Yaskawa INFORM job: KRIS7-TEST.JBI

/JOB
//NAME KRIS7-TEST
//POS
///NPOS 468,468,468,16,0,0
///TOOL 0
///POSTYPE PULSE
///PULSE
C00000=-36471,-76527,-106813,19264,71481,77238
C00001=-36471,-76527,-106813,19264,71481,77238
C00002=-63812,-119516,-80644,-27282,71106,59809
C00003=-86670,-29465,-24103,-33182,93398,46515
C00004=-88663,-31189,-25266,-33292,92471,45985
C00005=-89600,-31952,-25776,-33339,92036,45737
C00006=-88663,-31189,-25266,-33292,92471,45985
C00007=-88663,-31929,-28188,-33361,93666,45629
C00008=-101397,-33118,-34088,-22474,91022,41668
C00009=-101397,-32934,-33069,-22469,90527,41762
C00010=-101397,-33275,-35023,-22483,91481,41581
C00011=-104499,20623,14787,-23283,115207,62973
C00012=-104352,17765,12486,-23220,115200,63034
C00013=-104529,15851,10717,-23303,115245,62949
C00014=-104352,17765,12486,-23220,115200,63034
C00015=-100086,19810,13187,-22516,115799,63398
C00016=-93288,781,-1160,-33549,91987,44264
C00017=-95103,1586,-482,-33591,91265,43744
C00018=-95638,1156,-842,-33600,91054,43591
C00019=-95103,1586,-482,-33591,91265,43744
C00020=-100253,-3614,-11898,-25466,91372,41970
C00021=-107199,-8537,-17665,-19004,89460,40114
C00022=-108350,-8919,-17473,-17740,88760,39873
C00023=-102096,-5783,-13006,-25389,90415,41488
C00024=-93175,-13453,-24658,-25770,96080,43586
C00025=-29596,-126908,-80456,-16683,91164,67663
C00026=-130966,-130992,-81417,14801,93022,-34731
C00027=-139735,-123676,-71676,23223,79574,-40827
C00028=-136755,-124231,-71804,23689,78586,-39979
C00029=-134984,-124514,-71869,23951,78010,-39473
C00030=-136755,-124231,-71804,23689,78586,-39979
C00031=-136306,-124758,-74432,23664,79703,-39597
C00032=-105195,-127447,-79852,15126,73259,-28242
C00033=-104798,-126140,-77647,15190,72530,-28198
C00034=-108375,-128078,-79564,15067,73342,-29336
C00035=-112121,-93277,-65445,16297,96104,-47809
C00036=-116095,-84503,-58814,18813,102506,-48434
C00037=-114391,-86924,-59797,19239,101506,-47972
C00038=-116095,-84503,-58814,18813,102506,-48434
C00039=-117812,-129995,-81150,14641,74986,-32390
C00040=-118791,-92886,-67151,14205,85296,-31516
C00041=-116748,-92781,-67110,14299,84968,-30842
C00042=-115499,-92681,-67072,14351,84774,-30431
C00043=-116748,-92781,-67110,14299,84968,-30842
C00044=-116748,-94243,-70296,14285,86141,-30707
C00045=-102870,-92009,-70676,9222,86435,-25689
C00046=-102870,-90997,-68303,9229,85506,-25758
C00047=-102870,-92009,-70676,9222,86435,-25689
C00048=-124106,-98193,-79828,8318,91183,-32632
C00049=-120990,-117719,-86799,1028,78019,83969
C00050=-103618,-122878,-84450,6731,45671,69045
C00051=-107839,-39273,-43881,11021,86771,60654
C00052=-102663,-26959,-34255,5037,90909,61236
C00053=-106417,-22492,-30421,10624,98396,60708
C00054=-103076,-37240,-40581,8849,97261,61678
C00055=-110992,-39766,-43585,17340,97602,59383
C00056=-111851,-103912,-94699,10334,87868,68255
C00057=-100525,-93554,-87313,9422,87254,72087
C00058=-95765,-72558,-76889,7644,100510,59309
C00059=-95463,-76426,-71939,16938,115118,61391
C00060=-102124,-64154,-61473,23072,122501,60539
C00061=-108072,-63754,-61449,27079,123073,58329
C00062=-126453,-110744,-88068,25157,96958,85114
C00063=-124535,-114305,-86499,25277,93833,85163
C00064=-121951,-112497,-85625,25654,93398,86032
C00065=-116232,-108405,-84002,26384,92604,88006
C00066=-122754,-106725,-87203,25770,97209,86568
C00067=-142865,-91008,-85242,17891,113758,73123
C00068=-142005,-90205,-84914,18160,113770,73464
C00069=-93871,-48257,-54590,-14207,101968,-48555
C00070=-106716,17042,-5346,-15024,102835,-53222
C00071=-114740,-14345,-34597,-13608,101053,-59815
C00072=-127078,-3386,-21930,-8482,103399,-53955
C00073=-129021,-1243,-17298,-7607,102543,-53064
C00074=-129893,-13096,-22178,-14005,113849,-54571
C00075=-129597,-5294,-13720,-15224,118044,-55057
C00076=-122058,-3228,-13278,-23261,119236,-52777
C00077=-102997,28917,14853,-20600,116287,-84527
C00078=-102792,-6395,-13177,-23260,105514,-87254
C00079=-105472,-3384,-9862,-23514,105257,-88219
C00080=-107060,-2107,-8876,-23770,104848,-88744
C00081=-104416,1445,-8009,-23523,106791,-88129
C00082=-100743,5943,-9423,-11985,113108,-51981
C00083=-104100,-22795,-28366,-25068,61310,-50210
C00084=-122112,-33809,-21710,-17217,45375,-58941
C00085=-130767,-31374,-20493,-827,48037,-55558
C00086=-127443,-25046,-15801,-6227,47707,-53970
C00087=-124818,-6385,-1356,-9028,48013,-52772
C00088=-117469,-7945,-6130,-22808,51414,-49873
C00089=-27812,-119319,-87277,-42007,83182,-24370
C00090=-5621,-139291,-109992,-39952,96377,80222
C00091=-5621,-139291,-109992,-39952,96377,80222
C00092=87039,-115654,-82424,8022,52039,63522
C00093=129513,-144814,-136934,9080,53426,64546
C00094=125697,-42562,-22948,15669,36761,60413
C00095=126411,-45246,-5808,21270,25248,57573
C00096=137384,-94042,-14593,40484,4605,50802
C00097=156551,-106329,-15137,73999,-7456,40548
C00098=21972,-55240,6153,47914,22932,-29567
C00099=21236,-16271,22987,30471,58724,-17539
C00100=25572,-13994,24670,30139,57395,-16133
C00101=25572,-13994,24670,30139,57395,-16133
C00102=25572,-11360,29564,30679,55956,-16584
C00103=25572,-11642,29045,30620,56106,-16536
C00104=27131,-10690,29771,30483,55623,-16029
C00105=26687,-10968,29556,30524,55761,-16173
C00106=26687,-11435,28694,30427,56011,-16093
C00107=27498,-10924,29084,30350,55760,-15829
C00108=25574,-12112,28179,30521,56353,-16458
C00109=45065,-62251,-3802,30710,44756,-11744
C00110=45065,-62251,-3802,30710,44756,-11744
C00111=45062,-59455,603,31381,43658,-12167
C00112=45063,-59751,140,31308,43771,-12121
C00113=47363,-58455,705,30723,43318,-11195
C00114=46715,-58835,536,30894,43443,-11458
C00115=46717,-59324,-234,30775,43632,-11382
C00116=47899,-58629,71,30459,43407,-10903
C00117=45070,-60247,-636,31184,43956,-12046
C00118=91239,-86156,-11635,17290,26072,6257
C00119=91239,-86156,-11635,17290,26072,6257
C00120=91235,-83004,-7277,17966,25059,5922
C00121=91238,-83335,-7734,17887,25164,5961
C00122=92915,-81478,-7301,16273,25546,7147
C00123=92456,-82017,-7434,16717,25431,6822
C00124=92461,-82561,-8193,16597,25608,6883
C00125=93295,-81576,-7954,15794,25823,7471
C00126=91253,-83887,-8499,17745,25338,6030
C00127=158815,-84367,-11225,-29167,32105,45030
C00128=158815,-84367,-11225,-29167,32105,45030
C00129=158813,-81248,-6866,-30028,31158,45482
C00130=158816,-81574,-7323,-29937,31259,45435
C00131=156798,-79782,-6873,-28651,31269,44264
C00132=157356,-80302,-7010,-29015,31259,44592
C00133=157361,-80840,-7770,-28870,31430,44517
C00134=156355,-79886,-7523,-28212,31458,43925
C00135=158825,-82117,-8087,-29789,31433,45356
C00136=202470,-53277,302,-32057,53464,57737
C00137=202470,-53277,302,-32057,53464,57737
C00138=202470,-50579,4744,-32592,52316,58142
C00139=202471,-50863,4277,-32535,52437,58099
C00140=200347,-49670,4876,-32326,51937,57354
C00141=200948,-50019,4697,-32389,52078,57566
C00142=200949,-50488,3922,-32295,52282,57496
C00143=199855,-49845,4246,-32177,52030,57107
C00144=202472,-51331,3500,-32439,52645,58024
C00145=129513,-144814,-136934,9080,53426,64546
C00146=129513,-144814,-136934,9080,53426,64546
C00147=129513,-109632,-69732,14359,30578,61412
C00148=129513,-83278,-28536,22379,19314,57484
C00149=122399,-55102,-4999,-8402,35911,61097
C00150=119920,-45288,5620,-7331,30390,60229
C00151=119750,-46058,4611,-7150,30605,60108
C00152=119750,-45110,6218,-7257,30106,60163
C00153=119736,-46268,4531,-7151,30546,60106
C00154=119736,-47979,3777,-7238,30135,60151
C00155=119727,-46869,5444,-7329,29678,60198
C00156=119739,-46062,5830,-7299,29854,60181
C00157=119715,-47768,4014,-7231,30094,60141
C00158=122330,-55612,-6297,-8657,32618,61353
C00159=121709,-73745,-24049,9098,30676,53116
C00160=129398,-114812,-46545,3278,22913,57364
C00161=129398,-114812,-46545,3278,22913,57364
C00162=147189,-126166,-80752,5474,34460,60082
C00163=165214,-137669,-115409,7698,46160,62836
C00164=176409,-144814,-136934,9080,53426,64546
C00165=176409,-109327,-69248,14418,30440,61382
C00166=137996,-109327,-69248,14418,30440,61382
C00167=136854,5077,41656,21727,21645,57624
C00168=123203,14789,51546,53172,38991,40073
C00169=123077,34948,78392,59944,35543,36223
C00170=123077,37993,83408,61838,34770,35183
C00171=123098,35348,79007,60153,35442,36112
C00172=123139,31348,74887,59568,35673,36443
C00173=123149,34907,80133,61289,34946,35499
C00174=123130,37074,82445,61677,34805,35280
C00175=123183,30422,73312,58971,35912,36781
C00176=123599,57381,99984,51632,43856,40437
C00177=128629,59731,102899,52063,41097,41453
C00178=130023,30320,69348,52154,35987,38987
C00179=132104,19481,50493,23737,37003,47692
C00180=136200,48792,78585,9333,46433,53780
C00181=127667,43842,73216,11867,48213,50363
C00182=127110,36942,61073,12684,52130,50324
C00183=125174,17943,48073,21449,38985,45601
C00184=109988,7135,45797,56276,48109,34557
C00185=110783,-2370,26113,10588,43916,42309
C00186=96618,15106,36280,16308,48845,36588
C00187=99195,57631,83562,8929,54990,39222
C00188=83229,75338,108095,18392,45531,30732
C00189=82057,52050,70954,17595,54461,31693
C00190=99279,-29834,2408,12633,51480,38376
C00191=124602,-34297,-476,3581,48489,48797
C00192=129000,-155474,-110821,1722,53982,50766
C00193=129000,-186332,-136923,1718,54189,50769
C00194=129000,-186332,-136923,1718,54189,50769
C00195=124634,-42983,-17396,3288,54424,49011
C00196=119975,43106,65207,5416,48088,46799
C00197=124227,21838,45287,-4126,60993,49348
C00198=115102,22260,45694,-2630,60591,46004
C00199=111900,23179,46586,-2094,60423,44829
C00200=106599,25422,48781,-1196,60121,42879
C00201=109500,51617,73450,-2873,46958,44240
C00202=119708,-19564,1692,5024,54962,47046
C00203=124398,4257,31803,38326,49723,41965
C00204=124500,-5455,16693,36249,53145,43496
C00205=123978,22175,41893,32824,63757,46964
C00206=136633,26599,46213,31259,58773,50852
C00207=137127,47274,64261,33367,46328,47205
C00208=127043,-60461,-47717,31537,61680,47716
C00209=130427,-104246,-66216,34447,50964,45598
C00210=130427,-131180,-133049,27346,74705,52630
C00211=129293,-131648,-133187,27764,74930,52255
C00212=129293,-112975,-80869,32941,55210,46617
C00213=125224,-26758,-13299,33226,59088,46051
C00214=97492,-17863,6740,47317,62068,35221
C00215=76763,21057,43225,48272,71101,29312
C00216=80709,51150,75439,39481,73131,33496
C00217=101893,22474,45257,39781,66883,40263
C00218=98002,-1326,18556,46821,62661,35806
C00219=97492,-17863,6740,47317,62068,35221
C00220=125224,-26758,-13299,33226,59088,46051
C00221=129293,-131648,-133187,27764,74930,52255
C00222=129293,-130373,-135142,27565,76585,52657
C00223=129293,-130373,-135142,27565,76585,52657
C00224=129293,-130373,-135142,27565,76585,52657
C00225=126775,-65943,-41926,33631,56357,45828
C00226=146499,-5820,8509,-12483,47348,74367
C00227=133227,18598,33392,-5127,43166,68552
C00228=134087,40556,59352,-4333,44134,68757
C00229=109518,39473,58200,8432,44907,57480
C00230=110804,22133,33080,8574,45677,58038
C00231=95832,-100308,-60228,18401,42759,50383
C00232=85717,-180836,-128237,23276,45701,46095
C00233=134324,-194207,-130804,-6935,34984,69726
C00234=134324,-194207,-130804,-6935,34984,69726
C00235=134324,-194207,-130804,-6935,34984,69726
C00236=126554,-62104,-55568,-768,56192,65237
C00237=102691,-29899,-32559,11070,60126,55987
C00238=93699,-1684,15739,18283,46963,50224
C00239=95177,34388,59282,20423,38809,49091
C00240=95427,37375,44105,11480,58003,52927
C00241=82804,57701,66332,15963,56969,47713
C00242=80078,42075,52490,24500,50349,44630
C00243=92595,-4722,8571,18053,49920,50291
C00244=90890,13188,28851,45241,66990,53478
C00245=96516,51970,78121,48970,56932,51018
C00246=108766,35550,55769,36284,51974,56943
C00247=109501,48300,76470,39344,46724,54946
C00248=112089,47430,75488,38680,45769,55875
C00249=109461,35195,57508,36711,50675,56747
C00250=102961,43860,64049,37370,53600,54832
C00251=117347,37004,56694,33344,48695,60037
C00252=107165,27849,47408,45061,56134,56400
C00253=93699,-1684,15739,18283,46963,50224
C00254=126554,-62104,-55568,-768,56192,65237
C00255=132741,-190295,-136907,-5065,40605,68463
C00256=132741,-190295,-136907,-5065,40605,68463
C00257=132741,-190295,-136907,-5065,40605,68463
C00258=132741,-190295,-136907,-5065,40605,68463
C00259=126216,-48827,-32555,-652,48851,65144
C00260=116157,12397,26645,-836,43828,61032
C00261=107201,15073,29086,4732,43915,56787
C00262=108708,45240,59560,984,53519,57995
C00263=105889,47117,61614,1966,53270,56850
C00264=104117,15965,27840,6481,45345,55424
C00265=116157,12397,26645,-836,43828,61032
C00266=115184,32776,48658,-853,48273,60616
C00267=102009,39914,56094,5283,47719,54846
C00268=104295,38849,56164,-3583,45498,56420
C00269=106773,10666,21679,-1556,45201,57174
C00270=121513,8451,23347,32656,44981,60126
C00271=121479,33249,54130,32703,45073,60132
C00272=136244,38436,59676,26271,39414,66032
C00273=133358,13884,30500,26959,39421,64637
C00274=126216,-48827,-32555,-652,48851,65144
C00275=132741,-190295,-136907,-5065,40605,68463
C00276=132741,-190295,-136907,-5065,40605,68463
C00277=132741,-190295,-136907,-5065,40605,68463
C00278=132741,-190295,-136907,-5065,40605,68463
C00279=126554,-62104,-55568,-768,56192,65237
C00280=93699,-1684,15739,18283,46963,50224
C00281=109219,22842,33799,17593,55341,60017
C00282=114933,32716,55729,7970,41115,61622
C00283=98115,43367,67193,11592,40390,54327
C00284=92675,33947,50979,20393,49569,52577
C00285=113935,26100,44118,24451,47496,60162
C00286=114558,35388,59860,26260,42851,59091
C00287=117732,34768,59212,24806,41998,60459
C00288=114305,24559,43264,24398,47147,60243
C00289=99844,11402,27037,25299,53213,55440
C00290=126554,-62104,-55568,-768,56192,65237
C00291=132741,-190295,-136907,-5065,40605,68463
C00292=132741,-190295,-136907,-5065,40605,68463
C00293=132741,-190295,-136907,-5065,40605,68463
C00294=132741,-190295,-136907,-5065,40605,68463
C00295=126216,-48827,-32555,-652,48851,65144
C00296=134748,7082,18366,-200,46227,68791
C00297=132038,36511,51354,2924,49864,67481
C00298=110399,36003,50767,11764,51912,58463
C00299=101806,27679,40045,16592,51225,54569
C00300=102258,33237,49963,17192,48019,54198
C00301=104874,31614,48575,4374,45128,56525
C00302=106858,16986,29459,6761,48587,57166
C00303=113156,-2573,6178,11839,50347,59373
C00304=100847,-116604,-69788,21646,41420,51852
C00305=93537,-194381,-130385,26473,40988,47897
C00306=104459,-185785,-128899,13362,14722,54877
C00307=137185,-168918,-120422,-22616,31853,56508
C00308=103466,-143035,-89833,18127,44217,-664
C00309=153034,-42791,-3789,-574,51224,21077
C00310=154411,-23786,22188,6392,45845,11810
C00311=163692,-14831,30793,3045,43978,15753
C00312=162658,-12144,32796,3380,44162,15317
C00313=162658,-10372,35929,3443,43146,15280
C00314=162658,-10822,35136,3427,43403,15291
C00315=163644,-13399,33193,3102,43239,15709
C00316=163644,-12612,34572,3127,42795,15690
C00317=163043,-11060,35746,3327,42891,15434
C00318=163515,-12286,34819,3170,42815,15635
C00319=166152,-32133,5550,1997,50546,16952
C00320=100006,-46830,-3879,17345,57754,-8477
C00321=55652,-4276,24712,7053,56203,-22524
C00322=50070,19037,58848,16400,45172,-27179
C00323=51341,29328,71603,16783,42484,-27133
C00324=51341,32600,77102,17341,40853,-27469
C00325=51341,31422,75137,17137,41430,-27347
C00326=50264,28853,72458,17349,41942,-27728
C00327=50264,30492,75208,17635,41129,-27900
C00328=50738,31631,76404,17545,40896,-27733
C00329=50419,30858,75590,17605,41054,-27844
C00330=50419,14018,45638,14959,50461,-26136
C00331=53903,-12653,21571,13778,50962,-24612
C00332=66094,-67687,-18476,10677,45688,-20127
C00333=87454,-109874,-47340,-27972,40441,7116
C00334=78946,-55292,-6224,-23492,40558,2756
C00335=70027,-40972,10385,-20890,35738,-464
C00336=63439,-31094,22495,-18522,32104,-3061
C00337=63439,-29243,25592,-19018,31198,-2801
C00338=75556,-28394,37292,-62320,27769,16956
C00339=74155,-27422,37887,-61985,27131,16453
C00340=64318,-30449,24372,-21159,31089,-1672
C00341=67917,-25293,27676,-22824,32488,-51
C00342=67917,-25293,27676,-22824,32488,-51
C00343=68696,-24050,28500,-23162,32795,289
C00344=67917,-25293,27676,-22824,32488,-51
C00345=75368,-51805,-10970,-21451,43738,562
C00346=86139,-25078,5298,-24076,50017,4008
C00347=83917,-18337,16451,-24570,46284,3982
C00348=79836,-11066,25880,-23931,43276,2865
C00349=79836,-9413,28995,-24399,42297,3151
C00350=86314,-11086,32289,-42271,40319,10375
C00351=84998,-9998,33124,-41890,39785,9892
C00352=80963,-11349,26642,-26884,42529,4054
C00353=82363,-6834,30155,-27320,43093,4575
C00354=82761,-5465,31244,-27447,43243,4725
C00355=83186,-3958,32457,-27584,43396,4888
C00356=82761,-5465,31244,-27447,43243,4725
C00357=87385,-23200,183,-25112,53654,3858
C00358=88611,-6659,17671,-26227,51974,4862
C00359=85936,239,26154,-25964,49655,4281
C00360=85936,1480,28752,-26325,48787,4530
C00361=91127,630,32748,-40408,46738,9768
C00362=90313,1326,33333,-40211,46382,9497
C00363=86792,7,26768,-28149,49107,5083
C00364=90602,-33059,-4237,-28517,52203,5912
C00365=94576,-67258,-23025,57506,77870,-531
C00366=122383,-58832,-3556,65417,58097,774
C00367=127343,-13643,25366,63114,57669,4189
C00368=131296,13324,53885,65824,53660,3026
C00369=131296,14618,56173,66322,53341,2642
C00370=130824,14275,55697,67245,54004,2465
C00371=131723,14569,55971,67399,53464,2593
C00372=130860,14268,55674,67244,53987,2476
C00373=127124,-5804,29633,63377,58737,4694
C00374=126701,-15037,22522,63119,61223,3769
C00375=126701,1136,51385,68187,57095,-774
C00376=131284,6353,59362,70779,53649,-1335
C00377=131284,8754,63319,71617,53230,-1977
C00378=131284,6353,59362,70779,53649,-1335
C00379=132452,6685,59657,71098,52984,-1198
C00380=131284,6353,59362,70779,53649,-1335
C00381=131052,11501,64001,70861,53706,-1474
C00382=130893,14100,66417,70922,53742,-1574
C00383=130719,17099,69269,71021,53763,-1708
C00384=130893,14100,66417,70922,53742,-1574
C00385=128315,-22064,27147,66784,57381,941
C00386=129627,-37207,17556,68184,55855,186
C00387=130148,-23471,44300,74760,52317,-4741
C00388=135320,-14449,56479,79067,48853,-5949
C00389=135320,-12066,60154,79963,48630,-6563
C00390=135320,-14449,56479,79067,48853,-5949
C00391=137070,-14043,56767,79770,47945,-5809
C00392=135320,-14449,56479,79067,48853,-5949
C00393=134716,-10676,59212,78597,49226,-5841
C00394=134466,-8976,60486,78417,49378,-5807
C00395=134182,-6930,62050,78227,49545,-5776
C00396=134466,-8976,60486,78417,49378,-5807
C00397=106496,-51026,-9475,59829,73743,881
C00398=106496,-62277,-31108,58328,77765,3910
C00399=137468,-45448,-13164,23993,62707,9546
C00400=142031,-34381,-3630,18745,59946,9254
C00401=153480,-23481,18954,7895,48240,10284
C00402=154576,-15419,32985,7624,43640,10304
C00403=154522,-15140,33190,7639,43662,10282
C00404=163868,-10589,37972,6252,39486,12143
C00405=163705,-4288,45034,21073,38117,2051
C00406=163923,-2936,48273,26703,35302,170
C00407=146970,-27557,19782,29282,44621,-5055
C00408=77984,-28544,12598,9594,52255,-4511
C00409=87028,-14899,33509,-8097,43242,2023
C00410=86974,-14913,33498,-8080,43236,2001
C00411=77485,-7266,39372,-4959,42873,-2067
C00412=74579,-2521,47308,-17915,35684,548
C00413=75615,102,52227,-26296,32839,3633
C00414=84696,-19604,28451,-27180,39406,6073
C00415=87454,-109874,-47340,-27972,40441,7116
C00416=87454,-109874,-47340,-27972,40441,7116
C00417=73980,-36973,3355,-18473,60366,27525
C00418=58877,-27993,19766,-16405,50257,19650
C00419=71120,-6285,35203,-17245,53240,22132
C00420=69479,-8808,33067,-14788,50723,16894
C00421=73605,-31096,1389,-14177,59206,17320
C00422=72431,-18207,17991,-16956,51529,14828
C00423=73562,-15726,19761,-17396,52120,15565
C00424=83313,14185,44247,-21039,56473,22237
C00425=84211,-11070,13701,-18734,53182,26231
C00426=82998,-523,24465,-18637,51768,25979
C00427=82448,-570,28041,-15362,40529,26924
C00428=77134,-2165,39833,11119,14146,19838
C00429=76844,-12553,31864,7458,12108,20601
C00430=84341,-54767,463,-16268,10060,32559
C00431=79893,-46463,9240,-49361,8484,37720
C00432=71243,-22477,30789,30336,5200,-490
C00433=70979,-19028,33557,31433,5346,-1026
C00434=68683,-10375,50772,112552,4351,-37626
C00435=72976,-34040,25530,30096,2440,-170
C00436=51638,-47354,18402,88201,13764,-30312
C00437=50365,-30767,37744,101133,14655,-36527
C00438=46532,-17600,60099,119714,18815,-46088
C00439=50533,-52861,21550,106572,14840,-38992
C00440=66288,-93178,-46103,5866,60369,16168
C00441=112510,-98188,-44790,18471,62864,-44268
C00442=149625,-37879,6780,17046,57011,-35751
C00443=155605,-32525,16928,15112,50177,-29308
C00444=149418,-7594,34122,13784,51545,-27133
C00445=143716,-10385,36525,25765,46016,-27057
C00446=147766,-22217,9496,11268,57983,-23560
C00447=146875,-12758,20894,15319,55227,-24771
C00448=146053,-8471,24161,15451,55560,-25047
C00449=142035,19351,48051,16301,55907,-26583
C00450=141803,14161,44980,18392,51510,-21349
C00451=142040,5818,24378,13474,61789,-22474
C00452=138840,15265,37176,20739,58625,-24937
C00453=138706,17261,38894,20771,58629,-24991
C00454=139526,10572,40705,23596,37058,-29346
C00455=140566,11430,47120,26457,25355,-31911
C00456=140419,-8993,28489,25719,26277,-31573
C00457=142059,-17553,21658,25375,25949,-31323
C00458=143624,-11159,28730,24740,24544,-30775
C00459=144392,-5853,43056,31020,18891,-33660
C00460=150093,-42733,14524,24992,16002,-29807
C00461=146967,-32270,24662,40502,20136,-34953
C00462=144755,-20255,35089,33636,31779,-30408
C00463=144236,-61611,5153,41773,14596,-38681
C00464=136995,-150356,-85047,33892,64386,-36535
C00465=136995,-178339,-110283,33604,8697,-36217
C00466=130728,-161100,-136081,16173,33339,-28558
C00467=1271,-161100,-136081,16173,33339,-28558
BC00000=295325,674563,1075170
BC00001=295325,674563,1075170
BC00002=396971,731967,797664
BC00003=396971,731967,797664
BC00004=396971,731967,797664
BC00005=396971,731967,797664
BC00006=396971,731967,797664
BC00007=396971,731967,797664
BC00008=396971,731967,797664
BC00009=396971,731967,797664
BC00010=396971,731967,797664
BC00011=396971,731967,797664
BC00012=396971,731967,797664
BC00013=396971,731967,797664
BC00014=396971,731967,797664
BC00015=396971,731967,797664
BC00016=396971,731967,797664
BC00017=396971,731967,797664
BC00018=396971,731967,797664
BC00019=396971,731967,797664
BC00020=396971,731967,797664
BC00021=396971,731967,797664
BC00022=396971,731967,797664
BC00023=396971,731967,797664
BC00024=396971,731967,797664
BC00025=396971,731967,797664
BC00026=1331,731967,797664
BC00027=1331,834817,797664
BC00028=1331,834817,797664
BC00029=1331,834817,797664
BC00030=1331,834817,797664
BC00031=1331,834817,797664
BC00032=1331,834817,797664
BC00033=1331,834817,797664
BC00034=1331,834817,797664
BC00035=1331,834817,797664
BC00036=1331,834817,797664
BC00037=1331,834817,797664
BC00038=1331,834817,797664
BC00039=1331,834817,797664
BC00040=1331,834817,797664
BC00041=1331,834817,797664
BC00042=1331,834817,797664
BC00043=1331,834817,797664
BC00044=1331,834817,797664
BC00045=1331,834817,797664
BC00046=1331,834817,797664
BC00047=1331,834817,797664
BC00048=1331,834817,797664
BC00049=1072,761065,516765
BC00050=1072,827865,516765
BC00051=1071,829671,517043
BC00052=1071,829895,517078
BC00053=1071,829895,517078
BC00054=1071,829895,517078
BC00055=1071,829895,517078
BC00056=768,829895,695080
BC00057=768,829895,695080
BC00058=768,829895,695080
BC00059=768,829895,695080
BC00060=768,829895,695080
BC00061=768,829895,695080
BC00062=768,829895,695080
BC00063=768,829895,695080
BC00064=768,829895,695080
BC00065=768,829895,695080
BC00066=768,829895,695080
BC00067=768,829895,695080
BC00068=768,686767,695080
BC00069=396971,681851,797664
BC00070=396971,731967,797664
BC00071=396971,731967,797664
BC00072=396971,731967,797664
BC00073=396971,731967,797664
BC00074=396971,731967,797664
BC00075=396971,731967,797664
BC00076=396971,731967,797664
BC00077=396971,731967,797664
BC00078=396971,731967,797664
BC00079=396971,731967,797664
BC00080=396971,731967,797664
BC00081=396971,731967,797664
BC00082=396971,731967,797664
BC00083=396971,731967,516765
BC00084=396971,731967,516765
BC00085=396971,731967,516765
BC00086=396972,731979,516765
BC00087=396971,731967,516765
BC00088=396971,731967,516765
BC00089=396971,731967,516765
BC00090=188286,731967,1013423
BC00091=188286,774486,1052805
BC00092=125948,1177450,1071719
BC00093=215453,1309115,984509
BC00094=215453,1309115,984509
BC00095=215453,1269749,984509
BC00096=215453,1189879,984509
BC00097=215453,1164125,984509
BC00098=215453,1164125,984509
BC00099=215453,1164125,984509
BC00100=215453,1164125,984509
BC00101=215453,1164125,984509
BC00102=215453,1164125,984509
BC00103=215453,1164125,984509
BC00104=215453,1164125,984509
BC00105=215453,1164125,984509
BC00106=215453,1164125,984509
BC00107=215453,1164125,984509
BC00108=215453,1164125,984509
BC00109=215453,1164125,984509
BC00110=215453,1164125,984509
BC00111=215453,1164125,984509
BC00112=215453,1164125,984509
BC00113=215453,1164125,984509
BC00114=215453,1164125,984509
BC00115=215453,1164125,984509
BC00116=215453,1164125,984509
BC00117=215453,1164125,984509
BC00118=215453,1164125,984509
BC00119=215453,1164125,984509
BC00120=215453,1164125,984509
BC00121=215453,1164125,984509
BC00122=215453,1164125,984509
BC00123=215453,1164125,984509
BC00124=215453,1164125,984509
BC00125=215453,1164125,984509
BC00126=215453,1164125,984509
BC00127=215453,1164125,984509
BC00128=215453,1164125,984509
BC00129=215453,1164125,984509
BC00130=215453,1164125,984509
BC00131=215453,1164125,984509
BC00132=215453,1164125,984509
BC00133=215453,1164125,984509
BC00134=215453,1164125,984509
BC00135=215453,1164125,984509
BC00136=215453,1164125,984509
BC00137=215453,1164125,984509
BC00138=215453,1164125,984509
BC00139=215453,1164125,984509
BC00140=215453,1164125,984509
BC00141=215453,1164125,984509
BC00142=215453,1164125,984509
BC00143=215453,1164125,984509
BC00144=215453,1164125,984509
BC00145=215453,1309115,984509
BC00146=345399,1357897,984509
BC00147=345399,1357897,984509
BC00148=345399,1230997,984509
BC00149=346767,1230997,984506
BC00150=346767,1230997,984506
BC00151=346767,1230997,984506
BC00152=346767,1230997,984506
BC00153=346767,1230997,984506
BC00154=346767,1230997,984506
BC00155=346767,1230997,984506
BC00156=346767,1230997,984506
BC00157=346767,1230997,984506
BC00158=346767,1230997,984506
BC00159=309515,1253158,984507
BC00160=309515,1253158,984507
BC00161=309515,1328360,1051553
BC00162=314470,1361455,1064018
BC00163=253389,1357693,1050986
BC00164=215453,1309115,984509
BC00165=215453,1309115,984509
BC00166=135997,1309115,984509
BC00167=135997,1309115,984509
BC00168=135997,1309115,984509
BC00169=135997,1309115,984505
BC00170=135997,1309115,984505
BC00171=135997,1309115,984505
BC00172=135997,1309115,984505
BC00173=135997,1309115,984505
BC00174=135997,1309115,984505
BC00175=135997,1309115,984505
BC00176=135997,1309115,984509
BC00177=135997,1309115,984509
BC00178=135997,1309115,984509
BC00179=135997,1309115,984509
BC00180=135997,1309115,984509
BC00181=135997,1309115,984509
BC00182=135997,1309115,984509
BC00183=135997,1309115,984509
BC00184=135997,1309115,984509
BC00185=135997,1309115,984509
BC00186=94463,1309115,955550
BC00187=94463,1309115,963176
BC00188=94463,1309115,963176
BC00189=94463,1309115,963176
BC00190=94463,1309115,963176
BC00191=141941,1309115,963176
BC00192=141941,1309115,963176
BC00193=223116,1330631,963176
BC00194=328548,1330631,963176
BC00195=328548,1330631,963176
BC00196=328548,1330631,963176
BC00197=328548,1285890,963176
BC00198=328548,1285890,963176
BC00199=328548,1285890,963176
BC00200=328548,1285890,963176
BC00201=328548,1330631,963176
BC00202=328548,1291307,959498
BC00203=328548,1293601,963176
BC00204=328548,1288886,905196
BC00205=328548,1288886,905196
BC00206=328548,1288886,905196
BC00207=328824,1330631,905196
BC00208=328824,1330631,905196
BC00209=328824,1330631,905196
BC00210=328824,1330631,905196
BC00211=151003,1330631,905196
BC00212=151003,1330631,905196
BC00213=151003,1330631,905196
BC00214=103648,1289163,905196
BC00215=103648,1289163,905196
BC00216=103648,1289163,905196
BC00217=103648,1289163,905196
BC00218=103648,1289163,905196
BC00219=103648,1289163,905196
BC00220=151003,1330631,905196
BC00221=151003,1330631,905196
BC00222=151003,1330631,905196
BC00223=303803,1330631,905196
BC00224=303803,1330631,763831
BC00225=303803,1330631,902112
BC00226=303803,1330631,902112
BC00227=303803,1330631,902112
BC00228=303803,1330631,902112
BC00229=303803,1330631,902112
BC00230=303803,1330631,902112
BC00231=303803,1330631,902112
BC00232=303803,1330631,1003127
BC00233=236612,1330631,1003127
BC00234=137483,1330631,1003127
BC00235=136337,1325904,719417
BC00236=136337,1325904,818715
BC00237=87820,1325904,842743
BC00238=87820,1325904,951848
BC00239=87820,1325904,951848
BC00240=87820,1320020,844218
BC00241=87820,1320020,844218
BC00242=87820,1325904,927335
BC00243=87820,1325904,927335
BC00244=87820,1325904,927335
BC00245=87820,1325904,927335
BC00246=87820,1325904,927335
BC00247=87820,1325904,927335
BC00248=87820,1325904,927335
BC00249=87820,1325904,927335
BC00250=87820,1325904,890762
BC00251=87820,1325904,890392
BC00252=87820,1325904,927335
BC00253=87820,1325904,951848
BC00254=136337,1325904,818715
BC00255=136337,1325904,818715
BC00256=136337,1325904,998300
BC00257=310720,1325904,998300
BC00258=310720,1325904,777065
BC00259=310720,1325904,891809
BC00260=310720,1325904,891809
BC00261=310720,1325904,891809
BC00262=310720,1325904,891809
BC00263=310720,1325904,891809
BC00264=310720,1325904,891809
BC00265=310720,1325904,891809
BC00266=310720,1325904,891809
BC00267=310720,1325904,891809
BC00268=310720,1325904,891809
BC00269=310720,1325904,891809
BC00270=310720,1325904,891809
BC00271=310720,1325904,891809
BC00272=310720,1325904,891809
BC00273=310720,1325904,891809
BC00274=310720,1325904,891809
BC00275=310720,1325904,777065
BC00276=310720,1325904,998300
BC00277=136337,1325904,998300
BC00278=136337,1325904,818715
BC00279=136337,1325904,818715
BC00280=87820,1325904,951848
BC00281=87820,1325904,927335
BC00282=87820,1325904,927335
BC00283=87820,1325904,927335
BC00284=87820,1325904,927335
BC00285=87820,1325904,927335
BC00286=87820,1325904,927335
BC00287=87820,1325904,927335
BC00288=87820,1325904,927335
BC00289=87820,1325904,927335
BC00290=136337,1325904,818715
BC00291=136337,1325904,818715
BC00292=136337,1325904,998300
BC00293=310720,1325904,998300
BC00294=310720,1325904,777065
BC00295=310720,1325904,891809
BC00296=310720,1325904,891809
BC00297=310720,1325904,891809
BC00298=310720,1325904,891809
BC00299=310720,1325904,891809
BC00300=310720,1325904,891809
BC00301=310720,1325904,891809
BC00302=310720,1325904,891809
BC00303=310720,1325904,891809
BC00304=310720,1325904,891809
BC00305=310720,1325904,1051225
BC00306=230237,1331507,1051225
BC00307=214487,1257960,1051225
BC00308=187930,1133951,1051225
BC00309=187930,1063861,1051225
BC00310=187930,1063861,1051225
BC00311=187931,1063862,1051199
BC00312=187931,1063862,1051199
BC00313=187931,1063862,1051199
BC00314=187931,1063862,1051199
BC00315=187931,1063862,1051199
BC00316=187931,1063862,1051199
BC00317=187931,1063862,1051199
BC00318=187931,1063862,1051199
BC00319=187931,1063862,1051199
BC00320=187930,1063861,1051225
BC00321=187930,1063861,1051225
BC00322=187930,1063861,1051225
BC00323=187930,1063861,1051225
BC00324=187930,1063861,1051225
BC00325=187930,1063861,1051225
BC00326=187930,1063861,1051225
BC00327=187930,1063861,1051225
BC00328=187930,1063861,1051225
BC00329=187930,1063861,1051225
BC00330=187930,1063861,1051225
BC00331=187930,1063861,1051225
BC00332=187930,1063861,1051225
BC00333=244084,1125149,1051225
BC00334=244084,1125149,1051225
BC00335=244084,1125149,1051225
BC00336=244084,1125149,1051225
BC00337=244084,1125149,1051225
BC00338=244084,1125149,1051225
BC00339=244084,1125149,1051225
BC00340=244084,1125149,1051225
BC00341=244084,1125149,1051225
BC00342=244084,1125149,1051225
BC00343=244084,1125149,1051225
BC00344=244084,1125149,1051225
BC00345=244084,1125149,1051225
BC00346=244084,1125149,1051225
BC00347=244084,1125149,1051225
BC00348=244084,1125149,1051225
BC00349=244084,1125149,1051225
BC00350=244084,1125149,1051225
BC00351=244084,1125149,1051225
BC00352=244084,1125149,1051225
BC00353=244084,1125149,1051225
BC00354=244084,1125149,1051225
BC00355=244084,1125149,1051225
BC00356=244084,1125149,1051225
BC00357=244084,1125149,1051225
BC00358=244084,1125149,1051225
BC00359=244083,1125149,1051222
BC00360=244083,1125149,1051222
BC00361=244083,1125149,1051222
BC00362=244083,1125149,1051222
BC00363=244083,1125149,1051222
BC00364=244083,1125149,1051222
BC00365=244083,1125148,1051219
BC00366=166173,1125148,1051219
BC00367=166173,1125148,1051219
BC00368=166173,1142192,1051219
BC00369=166173,1142192,1051219
BC00370=166173,1142192,1051219
BC00371=166173,1142192,1051219
BC00372=166173,1142192,1051219
BC00373=166173,1142192,1051219
BC00374=166173,1142192,1051219
BC00375=166173,1142192,1051219
BC00376=166173,1142192,1051219
BC00377=166173,1142192,1051219
BC00378=166173,1142192,1051219
BC00379=166173,1142192,1051219
BC00380=166173,1142192,1051219
BC00381=166173,1142192,1051219
BC00382=166173,1142192,1051219
BC00383=166173,1142192,1051219
BC00384=166173,1142192,1051219
BC00385=166173,1142192,1051219
BC00386=166173,1142192,1051219
BC00387=166173,1142192,1051219
BC00388=166173,1142192,1051219
BC00389=166173,1142192,1051219
BC00390=166173,1142192,1051219
BC00391=166173,1142192,1051219
BC00392=166173,1142192,1051219
BC00393=166173,1142192,1051219
BC00394=166173,1142192,1051219
BC00395=166173,1142192,1051219
BC00396=166173,1142192,1051219
BC00397=166173,1142192,1051219
BC00398=166173,1142192,1051219
BC00399=180177,1091773,1051223
BC00400=182943,1081815,1051224
BC00401=187709,1064658,1051225
BC00402=187930,1063861,1051225
BC00403=187930,1063861,1051225
BC00404=187930,1063861,1051225
BC00405=187930,1063861,1051225
BC00406=187930,1063861,1051225
BC00407=187930,1063861,1051225
BC00408=244084,1063861,1051225
BC00409=244084,1063861,1051225
BC00410=244084,1063861,1051225
BC00411=244084,1063861,1051225
BC00412=244084,1063861,1051225
BC00413=244084,1063861,1051225
BC00414=244084,1063861,1051225
BC00415=244084,1063861,1051225
BC00416=244084,1125149,1051225
BC00417=244084,1125149,1051225
BC00418=244084,1125149,1051225
BC00419=244084,1125149,1051225
BC00420=244084,1125149,1051225
BC00421=244084,1125149,1051225
BC00422=244084,1125149,1051225
BC00423=244084,1125149,1051225
BC00424=244084,1125149,1051225
BC00425=244084,1125149,1051225
BC00426=244084,1125149,1051225
BC00427=244084,1125149,1051225
BC00428=244084,1125149,1051225
BC00429=244084,1125149,1051225
BC00430=244084,1125149,1051225
BC00431=244084,1125149,1051225
BC00432=244084,1125149,1051225
BC00433=244084,1125149,1051222
BC00434=244084,1125149,1051225
BC00435=244084,1125149,1051225
BC00436=244084,1125149,1051225
BC00437=244083,1125149,1051223
BC00438=244084,1125149,1051225
BC00439=244084,1125149,1051225
BC00440=244084,1125149,1051225
BC00441=148492,1125149,1051225
BC00442=148492,1157650,1055882
BC00443=148492,1157650,1055882
BC00444=148492,1157650,1055882
BC00445=148493,1157650,1055879
BC00446=148492,1157650,1055882
BC00447=148492,1157650,1055882
BC00448=148492,1157650,1055882
BC00449=148492,1157650,1055882
BC00450=148492,1157650,1055882
BC00451=148492,1157650,1055882
BC00452=148492,1157650,1055882
BC00453=148492,1157650,1055882
BC00454=148492,1157650,1055881
BC00455=148492,1157650,1055882
BC00456=148492,1157650,1055882
BC00457=148492,1157650,1055882
BC00458=148492,1157650,1055882
BC00459=148492,1157650,1055882
BC00460=148492,1157650,1055882
BC00461=148492,1157650,1055882
BC00462=148492,1157650,1055882
BC00463=148492,1157650,1055882
BC00464=148492,1157650,1055882
BC00465=189366,1229859,1070827
BC00466=189366,1118575,1070827
BC00467=189366,734808,1070827
EC00000=0,0
EC00001=-88685,-556476
EC00002=-88685,-556476
EC00003=-88685,-556476
EC00004=-88685,-556476
EC00005=-88685,-556476
EC00006=-88685,-556476
EC00007=-88685,-556476
EC00008=-88685,-556476
EC00009=-88685,-556476
EC00010=-88685,-556476
EC00011=-88685,-556476
EC00012=-88685,-556476
EC00013=-88685,-556476
EC00014=-88685,-556476
EC00015=-88685,-556476
EC00016=-88685,-556476
EC00017=-88685,-556476
EC00018=-88685,-556476
EC00019=-88685,-556476
EC00020=-88685,-556476
EC00021=-88685,-556476
EC00022=-88685,-556476
EC00023=-88685,-556476
EC00024=-88685,-556476
EC00025=-88685,-556476
EC00026=-88685,-556476
EC00027=-88685,-556476
EC00028=-88685,-556476
EC00029=-88685,-556476
EC00030=-88685,-556476
EC00031=-88685,-556476
EC00032=-88685,-556476
EC00033=-88685,-556476
EC00034=-88685,-556476
EC00035=-88685,-556476
EC00036=-88685,-556476
EC00037=-88685,-556476
EC00038=-88685,-556476
EC00039=-88685,-556476
EC00040=-88685,-556476
EC00041=-88685,-556476
EC00042=-88685,-556476
EC00043=-88685,-556476
EC00044=-88685,-556476
EC00045=-88685,-556476
EC00046=-88685,-556476
EC00047=-88685,-556476
EC00048=-88685,-556476
EC00049=264893,-556476
EC00050=264893,-556476
EC00051=264346,-556476
EC00052=264278,-556476
EC00053=264278,-556476
EC00054=264278,-556476
EC00055=264278,-556476
EC00056=-85879,-556476
EC00057=-85879,-556476
EC00058=-85879,-556476
EC00059=-85879,-556476
EC00060=-85879,-556476
EC00061=-85879,-556476
EC00062=-85879,-556476
EC00063=-85879,-556476
EC00064=-85879,-556476
EC00065=-85879,-556476
EC00066=-85879,-556476
EC00067=-85879,-556476
EC00068=-85879,-556476
EC00069=-88685,-556476
EC00070=-88685,-556476
EC00071=-88685,-612042
EC00072=-88685,-612042
EC00073=-88685,-612042
EC00074=-88685,-612042
EC00075=-88685,-612042
EC00076=-88685,-612042
EC00077=-88685,-556476
EC00078=-88685,-556476
EC00079=-88685,-556476
EC00080=-88685,-556476
EC00081=-88685,-556476
EC00082=-88685,-556476
EC00083=264893,-556476
EC00084=264893,-605076
EC00085=264893,-605076
EC00086=264894,-605076
EC00087=264893,-605076
EC00088=264893,-605076
EC00089=264893,-556476
EC00090=264890,-556476
EC00091=264890,-556476
EC00092=-210078,-556477
EC00093=-536455,-556477
EC00094=-536455,-556477
EC00095=-536455,-556477
EC00096=-536455,-556477
EC00097=-536455,-556477
EC00098=-536455,-556477
EC00099=-536455,-556477
EC00100=-536455,-556477
EC00101=-536455,-556477
EC00102=-536455,-556477
EC00103=-536455,-556477
EC00104=-536455,-556477
EC00105=-536455,-556477
EC00106=-536455,-556477
EC00107=-536455,-556477
EC00108=-536455,-556477
EC00109=-536455,-556477
EC00110=-536455,-556477
EC00111=-536455,-556477
EC00112=-536455,-556477
EC00113=-536455,-556477
EC00114=-536455,-556477
EC00115=-536455,-556477
EC00116=-536455,-556477
EC00117=-536455,-556477
EC00118=-536455,-556477
EC00119=-536455,-556477
EC00120=-536455,-556477
EC00121=-536455,-556477
EC00122=-536455,-556477
EC00123=-536455,-556477
EC00124=-536455,-556477
EC00125=-536455,-556477
EC00126=-536455,-556477
EC00127=-536455,-556477
EC00128=-536455,-556477
EC00129=-536455,-556477
EC00130=-536455,-556477
EC00131=-536455,-556477
EC00132=-536455,-556477
EC00133=-536455,-556477
EC00134=-536455,-556477
EC00135=-536455,-556477
EC00136=-536455,-556477
EC00137=-536455,-556477
EC00138=-536455,-556477
EC00139=-536455,-556477
EC00140=-536455,-556477
EC00141=-536455,-556477
EC00142=-536455,-556477
EC00143=-536455,-556477
EC00144=-536455,-556477
EC00145=-270405,-556477
EC00146=-270405,-556477
EC00147=-270405,-556477
EC00148=-270405,-556477
EC00149=-270404,-556477
EC00150=-270404,-556477
EC00151=-270404,-556477
EC00152=-270404,-556477
EC00153=-270404,-556477
EC00154=-270404,-556477
EC00155=-270404,-556477
EC00156=-270404,-556477
EC00157=-270404,-556477
EC00158=-270404,-556477
EC00159=-270404,-556477
EC00160=-270404,-556477
EC00161=-270404,-556477
EC00162=-270404,-556477
EC00163=-270405,-556477
EC00164=-270405,-556477
EC00165=-270405,-556477
EC00166=-270405,-556477
EC00167=-270405,-556477
EC00168=-270405,-556477
EC00169=-270404,-556477
EC00170=-270404,-556477
EC00171=-270404,-556477
EC00172=-270404,-556477
EC00173=-270404,-556477
EC00174=-270404,-556477
EC00175=-270404,-556477
EC00176=-270405,-556477
EC00177=-270405,-556477
EC00178=-270405,-556477
EC00179=-270405,-556477
EC00180=-270405,-556477
EC00181=-270405,-556477
EC00182=-270405,-556477
EC00183=-270405,-556477
EC00184=-270405,-556477
EC00185=-270405,-556477
EC00186=-270405,-556477
EC00187=-270405,-556477
EC00188=-270405,-556477
EC00189=-270405,-556477
EC00190=-270405,-556477
EC00191=-270405,-556477
EC00192=-270405,-556477
EC00193=-270405,-556477
EC00194=-270405,-556477
EC00195=-270405,-556477
EC00196=-270405,-556477
EC00197=-270405,-556477
EC00198=-270405,-556477
EC00199=-270405,-556477
EC00200=-270405,-556477
EC00201=-270405,-556477
EC00202=-270405,-556477
EC00203=-270405,-556477
EC00204=-270405,-556477
EC00205=-270405,-556477
EC00206=-270405,-556477
EC00207=-270405,-556477
EC00208=-270405,-556477
EC00209=-270405,-556477
EC00210=-270405,-556477
EC00211=-270405,-556477
EC00212=-270405,-556477
EC00213=-270405,-556477
EC00214=-270405,-556477
EC00215=-270405,-556477
EC00216=-270405,-556477
EC00217=-270405,-556477
EC00218=-270405,-556477
EC00219=-270405,-556477
EC00220=-270405,-556477
EC00221=-270405,-556477
EC00222=-270405,-556477
EC00223=-270405,-556477
EC00224=-270405,-556477
EC00225=-270405,-556477
EC00226=-270405,-556477
EC00227=-270405,-556477
EC00228=-270405,-556477
EC00229=-270405,-556477
EC00230=-270405,-556477
EC00231=-270405,-556477
EC00232=-270405,-556477
EC00233=-270405,-556477
EC00234=-270405,-556477
EC00235=-270405,-556477
EC00236=-270405,-556477
EC00237=-270405,-556477
EC00238=-270405,-556477
EC00239=-270405,-556477
EC00240=-270405,-556477
EC00241=-270405,-556477
EC00242=-270405,-556477
EC00243=-270405,-556477
EC00244=-270405,-556477
EC00245=-270405,-556477
EC00246=-270405,-556477
EC00247=-270405,-556477
EC00248=-270405,-556477
EC00249=-270405,-556477
EC00250=-270405,-556477
EC00251=-270405,-556477
EC00252=-270405,-556477
EC00253=-270405,-556477
EC00254=-270405,-556477
EC00255=-270405,-556477
EC00256=-270405,-556477
EC00257=-270405,-556477
EC00258=-270405,-556477
EC00259=-270405,-556477
EC00260=-270405,-556477
EC00261=-270405,-556477
EC00262=-270405,-556477
EC00263=-270405,-556477
EC00264=-270405,-556477
EC00265=-270405,-556477
EC00266=-270405,-556477
EC00267=-270405,-556477
EC00268=-270405,-556477
EC00269=-270405,-556477
EC00270=-270405,-556477
EC00271=-270405,-556477
EC00272=-270405,-556477
EC00273=-270405,-556477
EC00274=-270405,-556477
EC00275=-270405,-556477
EC00276=-270405,-556477
EC00277=-270405,-556477
EC00278=-270405,-556477
EC00279=-270405,-556477
EC00280=-270405,-556477
EC00281=-270405,-556477
EC00282=-270405,-556477
EC00283=-270405,-556477
EC00284=-270405,-556477
EC00285=-270405,-556477
EC00286=-270405,-556477
EC00287=-270405,-556477
EC00288=-270405,-556477
EC00289=-270405,-556477
EC00290=-270405,-556477
EC00291=-270405,-556477
EC00292=-270405,-556477
EC00293=-270405,-556477
EC00294=-270405,-556477
EC00295=-270405,-556477
EC00296=-270405,-556477
EC00297=-270405,-556477
EC00298=-270405,-556477
EC00299=-270405,-556477
EC00300=-270405,-556477
EC00301=-270405,-556477
EC00302=-270405,-556477
EC00303=-270405,-556477
EC00304=-270405,-556477
EC00305=-270405,-556477
EC00306=-270405,-556477
EC00307=-270405,-556477
EC00308=-270405,-556477
EC00309=-270405,-556477
EC00310=-270405,-556477
EC00311=-270402,-556478
EC00312=-270402,-556478
EC00313=-270402,-556478
EC00314=-270402,-556478
EC00315=-270402,-556478
EC00316=-270402,-556478
EC00317=-270402,-556478
EC00318=-270402,-556478
EC00319=-270402,-556478
EC00320=-270405,-556477
EC00321=-270405,-556477
EC00322=-270405,-556477
EC00323=-270405,-556477
EC00324=-270405,-556477
EC00325=-270405,-556477
EC00326=-270405,-556477
EC00327=-270405,-556477
EC00328=-270405,-556477
EC00329=-270405,-556477
EC00330=-270405,-556477
EC00331=-270405,-556477
EC00332=-270405,-556477
EC00333=-447795,-556477
EC00334=-447795,-556477
EC00335=-447795,-556477
EC00336=-447795,-556477
EC00337=-447795,-556477
EC00338=-447795,-556477
EC00339=-447795,-556477
EC00340=-447795,-556477
EC00341=-447795,-556477
EC00342=-447795,-556477
EC00343=-447795,-556477
EC00344=-447795,-556477
EC00345=-447795,-556477
EC00346=-447795,-556477
EC00347=-447795,-556477
EC00348=-447795,-556477
EC00349=-447795,-556477
EC00350=-447795,-556477
EC00351=-447795,-556477
EC00352=-447795,-556477
EC00353=-447795,-556477
EC00354=-447795,-556477
EC00355=-447795,-556477
EC00356=-447795,-556477
EC00357=-447795,-556477
EC00358=-447795,-556477
EC00359=-447793,-556477
EC00360=-447793,-556477
EC00361=-447793,-556477
EC00362=-447793,-556477
EC00363=-447793,-556477
EC00364=-447793,-556477
EC00365=-447791,-556477
EC00366=-447791,-556477
EC00367=-447791,-556477
EC00368=-447791,-556477
EC00369=-447791,-556477
EC00370=-447791,-556477
EC00371=-447791,-556477
EC00372=-447791,-556477
EC00373=-447791,-556477
EC00374=-447791,-556477
EC00375=-447791,-556477
EC00376=-447791,-556477
EC00377=-447791,-556477
EC00378=-447791,-556477
EC00379=-447791,-556477
EC00380=-447791,-556477
EC00381=-447791,-556477
EC00382=-447791,-556477
EC00383=-447791,-556477
EC00384=-447791,-556477
EC00385=-447791,-556477
EC00386=-447791,-556477
EC00387=-447791,-556477
EC00388=-447791,-556477
EC00389=-447791,-556477
EC00390=-447791,-556477
EC00391=-447791,-556477
EC00392=-447791,-556477
EC00393=-447791,-556477
EC00394=-447791,-556477
EC00395=-447791,-556477
EC00396=-447791,-556477
EC00397=-447791,-556477
EC00398=-447791,-556477
EC00399=-333615,-556477
EC00400=-311064,-556477
EC00401=-272209,-556477
EC00402=-270405,-556477
EC00403=-270405,-556477
EC00404=-270405,-556477
EC00405=-270405,-556477
EC00406=-270405,-556477
EC00407=-270405,-556477
EC00408=-270405,-556477
EC00409=-270405,-556477
EC00410=-270405,-556477
EC00411=-270405,-556477
EC00412=-270405,-556477
EC00413=-270405,-556477
EC00414=-270405,-556477
EC00415=-270405,-556477
EC00416=-447795,-556477
EC00417=-447795,-556477
EC00418=-447795,-556477
EC00419=-447795,-556477
EC00420=-447795,-556477
EC00421=-447795,-556477
EC00422=-447795,-556477
EC00423=-447795,-556477
EC00424=-447795,-556477
EC00425=-447795,-556477
EC00426=-447795,-556477
EC00427=-447795,-556477
EC00428=-447795,-556477
EC00429=-447795,-556477
EC00430=-447795,-556477
EC00431=-447795,-556477
EC00432=-447795,-556477
EC00433=-447794,-556477
EC00434=-447795,-556477
EC00435=-447795,-556477
EC00436=-447795,-556477
EC00437=-447794,-556478
EC00438=-447795,-556477
EC00439=-447795,-556477
EC00440=-447795,-556477
EC00441=-447795,-556477
EC00442=-447795,-556477
EC00443=-447795,-556477
EC00444=-447795,-556477
EC00445=-447793,-556477
EC00446=-447795,-556477
EC00447=-447795,-556477
EC00448=-447795,-556477
EC00449=-447795,-556477
EC00450=-447795,-556477
EC00451=-447795,-556477
EC00452=-447795,-556477
EC00453=-447795,-556477
EC00454=-447794,-556478
EC00455=-447795,-556477
EC00456=-447795,-556477
EC00457=-447795,-556477
EC00458=-447795,-556477
EC00459=-447795,-556477
EC00460=-447795,-556477
EC00461=-447795,-556477
EC00462=-447795,-556477
EC00463=-447795,-556477
EC00464=-447795,-556477
EC00465=-447795,-556477
EC00466=-71624,-556477
EC00467=15446,-556477
///POSTYPE BASE
///RECTAN
///RCONF 0,0,0,0,0,0,0,0,0,0,0,0,0,0,0,0,0,0,0,0,0,0,0,0
P00006=0.000,0.000,0.000,0.0000,0.0000,0.0000
P00032=1.957,0.503,-7.217,0.0000,0.0000,0.0000
///RCONF 0,0,0,0,1,0,0,0,0,0,0,0,0,0,0,0,0,0,0,0,0,0,0,0
P00033=-0.123,0.612,-5.012,0.0000,0.0000,0.0000
///RCONF 0,0,0,0,0,0,0,0,0,0,0,0,0,0,0,0,0,0,0,0,0,0,0,0
P00034=-0.304,0.773,-2.693,0.0000,0.0000,0.0000
P00035=2.817,0.591,-1.622,0.0000,0.0000,0.0000
P00040=-0.030,9.648,2.467,0.0000,0.0000,0.0000
P00041=0.192,3.924,0.305,0.0000,0.0000,0.0000
P00042=-0.217,1.941,0.413,0.0000,0.0000,0.0000
P00043=-0.044,-1.937,1.197,0.0000,0.0000,0.0000
P00044=0.687,-2.322,1.156,0.0000,0.0000,0.0000
P00045=-0.068,-0.810,1.603,0.0000,0.0000,0.0000
P00046=0.799,0.043,1.292,0.0000,0.0000,0.0000
///RCONF 0,1,0,0,0,0,0,0,0,0,0,0,0,0,0,0,0,0,0,0,0,0,0,0
P00047=-0.011,1.737,-0.646,0.0000,0.0000,0.0000
///RCONF 0,0,0,0,0,0,0,0,0,0,0,0,0,0,0,0,0,0,0,0,0,0,0,0
P00048=2.411,0.025,-0.606,0.0000,0.0000,0.0000
P00049=3.413,-3.572,-1.618,0.0000,0.0000,0.0000
P00050=4.296,-4.501,-0.826,0.0000,0.0000,0.0000
//INST
///DATE 2025/01/08 12:13
///ATTR SC,RW
///GROUP1 RB1,BS1
///GROUP2 ST1
NOP
MOVJ C00000 BC00000 VJ=100.00  +MOVJ EC00000 VJ=100.00
MOVJ C00001 BC00001 VJ=100.00  +MOVJ EC00001 VJ=100.00
CALL JOB:CLEAN-R1_KM_NEW
MOVJ C00002 BC00002 VJ=100.00  +MOVJ EC00002 VJ=100.00
MOVJ C00003 BC00003 VJ=50.00  +MOVJ EC00003 VJ=50.00
SMOVL C00004 BC00004 V=83.3  +MOVJ EC00004
SREFP 3 C00005 BC00005  +REFP EC00005
CALL JOB:SEARCH-R1-S13D
SET P032 P006
SFTON3D P032
SMOVL C00006 BC00006 V=60.0  +MOVJ EC00006
SMOVL C00007 BC00007 V=133.3  +MOVJ EC00007
SMOVL C00008 BC00008 V=133.3  +MOVJ EC00008
SREFP 3 C00009 BC00009  +REFP EC00009
CALL JOB:SEARCH-R1-S13D
SET P032 P006
SFTON3D P032
SMOVL C00010 BC00010 V=60.0  +MOVJ EC00010
SMOVL C00011 BC00011 V=133.3  +MOVJ EC00011
SMOVL C00012 BC00012 V=133.3  +MOVJ EC00012
SREFP 3 C00013 BC00013  +REFP EC00013
CALL JOB:SEARCH-R1-S13D
SET P032 P006
SFTON3D P032
SFTOF3D
SMOVL C00014 BC00014 V=133.3  +MOVJ EC00014
SMOVL C00015 BC00015 V=200.0  +MOVJ EC00015
SFTOF3D
'S1
MOVJ C00016 BC00016 VJ=50.00  +MOVJ EC00016 VJ=50.00
'S2
SMOVL C00017 BC00017 V=60.0  +MOVJ EC00017
SREFP 3 C00018 BC00018  +REFP EC00018
CALL JOB:SEARCH-R1-S13D
SET P033 P006
SFTON3D P033
SMOVL C00019 BC00019 V=60.0  +MOVJ EC00019
SMOVL C00020 BC00020 V=133.3  +MOVJ EC00020
SMOVL C00021 BC00021 V=133.3  +MOVJ EC00021
SREFP 3 C00022 BC00022  +REFP EC00022
CALL JOB:SEARCH-R1-S13D
SET P033 P006
SFTON3D P033
SFTOF3D
SMOVL C00023 BC00023 V=83.3  +MOVJ EC00023
MOVJ C00024 BC00024 VJ=60.00  +MOVJ EC00024 VJ=60.00
MOVJ C00025 BC00025 VJ=60.00  +MOVJ EC00025 VJ=60.00
MOVJ C00026 BC00026 VJ=100.00  +MOVJ EC00026 VJ=60.00
MOVJ C00027 BC00027 VJ=60.00  +MOVJ EC00027 VJ=60.00
SMOVL C00028 BC00028 V=60.0  +MOVJ EC00028
SREFP 3 C00029 BC00029  +REFP EC00029
CALL JOB:SEARCH-R1-S13D
SET P034 P006
SFTON3D P034
SMOVL C00030 BC00030 V=60.0  +MOVJ EC00030
SMOVL C00031 BC00031 V=83.3  +MOVJ EC00031
SMOVL C00032 BC00032 V=83.3  +MOVJ EC00032
SREFP 3 C00033 BC00033  +REFP EC00033
CALL JOB:SEARCH-R1-S13D
SET P034 P006
SFTON3D P034
SMOVL C00034 BC00034 V=100.0  +MOVJ EC00034
SMOVL C00035 BC00035 V=133.3  +MOVJ EC00035
SMOVL C00036 BC00036 V=133.3  +MOVJ EC00036
SREFP 3 C00037 BC00037  +REFP EC00037
CALL JOB:SEARCH-R1-S13D
SET P034 P006
SFTON3D P034
SMOVL C00038 BC00038 V=133.3  +MOVJ EC00038
SMOVL C00039 BC00039 V=133.3  +MOVJ EC00039
SMOVL C00040 BC00040 V=250.0  +MOVJ EC00040
SMOVL C00041 BC00041 V=60.0  +MOVJ EC00041
SREFP 3 C00042 BC00042  +REFP EC00042
CALL JOB:SEARCH-R1-S13D
SET P035 P006
SFTON3D P035
SMOVL C00043 BC00043 V=60.0  +MOVJ EC00043
SMOVL C00044 BC00044 V=250.0  +MOVJ EC00044
SMOVL C00045 BC00045 V=250.0  +MOVJ EC00045
SREFP 3 C00046 BC00046  +REFP EC00046
CALL JOB:SEARCH-R1-S13D
SET P035 P006
SFTON3D P035
SMOVL C00047 BC00047 V=166.7  +MOVJ EC00047
SFTOF3D
MOVJ C00048 BC00048 VJ=30.00  +MOVJ EC00048 VJ=15.00
MOVJ C00049 BC00049 VJ=100.00  +MOVJ EC00049 VJ=50.00
MACRO1 MJ#(0) ARGF9
MOVJ C00050 BC00050 VJ=100.00  +MOVJ EC00050 VJ=15.00
SMOVL C00051 BC00051 V=666.7  +MOVJ EC00051
SFTON3D P035
SMOVL C00052 BC00052 V=166.7  +MOVJ EC00052
ARCON
SMOVL C00053 BC00053 V=6.7  +MOVJ EC00053
SMOVL C00054 BC00054 V=6.7  +MOVJ EC00054
ARCOF
TIMER T=1.00
SMOVL C00055 BC00055 V=166.7  +MOVJ EC00055
SFTOF3D
MOVJ C00056 BC00056 VJ=100.00  +MOVJ EC00056 VJ=100.00
MOVJ C00057 BC00057 VJ=15.00  +MOVJ EC00057 VJ=100.00
SFTON3D P035
SMOVL C00058 BC00058 V=166.7  +MOVJ EC00058
ARCON
SFTON3D P034
SMOVL C00059 BC00059 V=8.3  +MOVJ EC00059
SMOVL C00060 BC00060 V=8.3  +MOVJ EC00060
ARCOF
SMOVL C00061 BC00061 V=166.7  +MOVJ EC00061
SMOVL C00062 BC00062 V=500.0  +MOVJ EC00062
SMOVL C00063 BC00063 V=166.7  +MOVJ EC00063
ARCON
SMOVL C00064 BC00064 V=7.5  +MOVJ EC00064
SMOVL C00065 BC00065 V=7.5  +MOVJ EC00065
ARCOF
SFTOF3D
MOVJ C00066 BC00066 VJ=30.00  +MOVJ EC00066 VJ=60.00
MOVJ C00067 BC00067 VJ=100.00  +MOVJ EC00067 VJ=50.00
MOVJ C00068 BC00068 VJ=100.00  +MOVJ EC00068 VJ=15.00
MOVJ C00069 BC00069 VJ=100.00  +MOVJ EC00069 VJ=100.00
MOVJ C00070 BC00070 VJ=50.00  +MOVJ EC00070 VJ=50.00
SFTOF3D
MOVJ C00071 BC00071 VJ=100.00  +MOVJ EC00071 VJ=100.00
MOVJ C00072 BC00072 VJ=100.00  +MOVJ EC00072 VJ=100.00
SFTON3D P033
SMOVL C00073 BC00073 V=166.7  +MOVJ EC00073
ARCON
SFTON3D P032
SMOVL C00074 BC00074 V=8.3  +MOVJ EC00074
SMOVL C00075 BC00075 V=8.3  +MOVJ EC00075
ARCOF
SMOVL C00076 BC00076 V=166.7  +MOVJ EC00076
SMOVL C00077 BC00077 V=666.7  +MOVJ EC00077
SMOVL C00078 BC00078 V=133.3  +MOVJ EC00078
ARCON
SMOVL C00079 BC00079 V=7.5  +MOVJ EC00079
SMOVL C00080 BC00080 V=7.5  +MOVJ EC00080
ARCOF
SFTOF3D
SMOVL C00081 BC00081 V=133.3  +MOVJ EC00081
MOVJ C00082 BC00082 VJ=50.00  +MOVJ EC00082 VJ=50.00
MOVJ C00083 BC00083 VJ=100.00  +MOVJ EC00083 VJ=100.00
MOVJ C00084 BC00084 VJ=100.00  +MOVJ EC00084 VJ=100.00
SFTON3D P033
SMOVL C00085 BC00085 V=133.3  +MOVJ EC00085
ARCON
SMOVL C00086 BC00086 V=7.5  +MOVJ EC00086
ARCON
SMOVL C00087 BC00087 V=7.5  +MOVJ EC00087
ARCOF
MOVJ C00088 BC00088 VJ=50.00  +MOVJ EC00088 VJ=50.00
MOVJ C00089 BC00089 VJ=100.00  +MOVJ EC00089 VJ=100.00
CALL JOB:CLEAN-R1_KM_NEW
MOVJ C00090 BC00090 VJ=100.00  +MOVJ EC00090 VJ=100.00
MOVJ C00091 BC00091 VJ=100.00  +MOVJ EC00091 VJ=100.00
MOVJ C00092 BC00092 VJ=100.00  +MOVJ EC00092 VJ=100.00
PAUSE
MOVJ C00093 BC00093 VJ=100.00  +MOVJ EC00093 VJ=100.00
MOVJ C00094 BC00094 VJ=100.00  +MOVJ EC00094 VJ=100.00
MOVJ C00095 BC00095 VJ=100.00  +MOVJ EC00095 VJ=100.00
MOVJ C00096 BC00096 VJ=100.00  +MOVJ EC00096 VJ=100.00
MOVJ C00097 BC00097 VJ=100.00  +MOVJ EC00097 VJ=100.00
MOVL C00098 BC00098 V=666.7  +MOVJ EC00098 VJ=100.00
MOVL C00099 BC00099 V=333.3  +MOVJ EC00099 VJ=100.00
MOVL C00100 BC00100 V=333.3  +MOVJ EC00100 VJ=100.00
SMOVL C00101 BC00101 V=100.0  +MOVJ EC00101
SREFP 3 C00102 BC00102  +REFP EC00102
CALL JOB:SEARCH-R1-S13D
SET P041 P006
SFTON3D P041
SMOVL C00103 BC00103 V=166.7  +MOVJ EC00103
SREFP 3 C00104 BC00104  +REFP EC00104
CALL JOB:SEARCH-R1-S13D
SET P041 P006
SFTON3D P041
SMOVL C00105 BC00105 V=166.7  +MOVJ EC00105
SMOVL C00106 BC00106 V=166.7  +MOVJ EC00106
SREFP 3 C00107 BC00107  +REFP EC00107
CALL JOB:SEARCH-R1-S13D
SET P042 P006
SFTON3D P042
SMOVL C00108 BC00108 V=166.7  +MOVJ EC00108
MOVL C00109 BC00109 V=333.3  +MOVJ EC00109 VJ=100.00
SMOVL C00110 BC00110 V=100.0  +MOVJ EC00110
SREFP 3 C00111 BC00111  +REFP EC00111
CALL JOB:SEARCH-R1-S13D
SET P043 P006
SFTON3D P043
SMOVL C00112 BC00112 V=166.7  +MOVJ EC00112
SREFP 3 C00113 BC00113  +REFP EC00113
CALL JOB:SEARCH-R1-S13D
SET P043 P006
SFTON3D P043
SMOVL C00114 BC00114 V=166.7  +MOVJ EC00114
SMOVL C00115 BC00115 V=166.7  +MOVJ EC00115
SREFP 3 C00116 BC00116  +REFP EC00116
CALL JOB:SEARCH-R1-S13D
SET P044 P006
SFTON3D P044
SMOVL C00117 BC00117 V=166.7  +MOVJ EC00117
MOVL C00118 BC00118 V=333.3  +MOVJ EC00118 VJ=100.00
SMOVL C00119 BC00119 V=100.0  +MOVJ EC00119
SREFP 3 C00120 BC00120  +REFP EC00120
CALL JOB:SEARCH-R1-S13D
SET P045 P006
SFTON3D P045
SMOVL C00121 BC00121 V=166.7  +MOVJ EC00121
SREFP 3 C00122 BC00122  +REFP EC00122
CALL JOB:SEARCH-R1-S13D
SET P045 P006
SFTON3D P045
SMOVL C00123 BC00123 V=166.7  +MOVJ EC00123
SMOVL C00124 BC00124 V=166.7  +MOVJ EC00124
SREFP 3 C00125 BC00125  +REFP EC00125
CALL JOB:SEARCH-R1-S13D
SET P046 P006
SFTON3D P046
SMOVL C00126 BC00126 V=166.7  +MOVJ EC00126
MOVL C00127 BC00127 V=333.3  +MOVJ EC00127 VJ=100.00
SMOVL C00128 BC00128 V=100.0  +MOVJ EC00128
SREFP 3 C00129 BC00129  +REFP EC00129
CALL JOB:SEARCH-R1-S13D
SET P047 P006
SFTON3D P047
SMOVL C00130 BC00130 V=166.7  +MOVJ EC00130
SREFP 3 C00131 BC00131  +REFP EC00131
CALL JOB:SEARCH-R1-S13D
SET P047 P006
SFTON3D P047
SMOVL C00132 BC00132 V=166.7  +MOVJ EC00132
SMOVL C00133 BC00133 V=166.7  +MOVJ EC00133
SREFP 3 C00134 BC00134  +REFP EC00134
CALL JOB:SEARCH-R1-S13D
SET P048 P006
SFTON3D P048
SMOVL C00135 BC00135 V=166.7  +MOVJ EC00135
MOVL C00136 BC00136 V=333.3  +MOVJ EC00136 VJ=100.00
SMOVL C00137 BC00137 V=100.0  +MOVJ EC00137
SREFP 3 C00138 BC00138  +REFP EC00138
CALL JOB:SEARCH-R1-S13D
SET P049 P006
SFTON3D P049
SMOVL C00139 BC00139 V=166.7  +MOVJ EC00139
SREFP 3 C00140 BC00140  +REFP EC00140
CALL JOB:SEARCH-R1-S13D
SET P049 P006
SFTON3D P049
SMOVL C00141 BC00141 V=166.7  +MOVJ EC00141
SMOVL C00142 BC00142 V=166.7  +MOVJ EC00142
SREFP 3 C00143 BC00143  +REFP EC00143
CALL JOB:SEARCH-R1-S13D
SET P050 P006
SFTON3D P050
SMOVL C00144 BC00144 V=166.7  +MOVJ EC00144
PAUSE
COMM MOVJ C00145 BC00145 VJ=100.00  +MOVJ EC00145 VJ=50.00
COMM MOVJ C00146 BC00146 VJ=100.00  +MOVJ EC00146 VJ=50.00
COMM MOVJ C00147 BC00147 VJ=100.00  +MOVJ EC00147 VJ=50.00
COMM MOVJ C00148 BC00148 VJ=100.00  +MOVJ EC00148 VJ=50.00
COMM MOVJ C00149 BC00149 VJ=100.00  +MOVJ EC00149 VJ=15.00
COMM SFTOF3D
COMM MOVJ C00150 BC00150 VJ=15.00  +MOVJ EC00150 VJ=15.00
COMM SMOVL C00151 BC00151 V=100.0  +MOVJ EC00151
COMM SREFP 3 C00152 BC00152  +REFP EC00152
COMM CALL JOB:SEARCH-R1-S13D
COMM SET P041 P006
COMM SFTON3D P041
COMM SMOVL C00153 BC00153 V=100.0  +MOVJ EC00153
COMM SMOVL C00154 BC00154 V=83.3  +MOVJ EC00154
COMM SMOVL C00155 BC00155 V=83.3  +MOVJ EC00155
COMM SREFP 3 C00156 BC00156  +REFP EC00156
COMM CALL JOB:SEARCH-R1-S13D
COMM SET P041 P006
COMM SFTON3D P041
COMM SMOVL C00157 BC00157 V=100.0  +MOVJ EC00157
COMM SFTOF3D
COMM MOVJ C00158 BC00158 VJ=40.00  +MOVJ EC00158 VJ=100.00
COMM MOVJ C00159 BC00159 VJ=100.00  +MOVJ EC00159 VJ=15.00
COMM MOVJ C00160 BC00160 VJ=100.00  +MOVJ EC00160 VJ=15.00
COMM MOVJ C00161 BC00161 VJ=100.00  +MOVJ EC00161 VJ=15.00
COMM MOVJ C00162 BC00162 VJ=100.00  +MOVJ EC00162 VJ=15.00
COMM MOVJ C00163 BC00163 VJ=30.00  +MOVJ EC00163 VJ=15.00
COMM MOVJ C00164 BC00164 VJ=100.00  +MOVJ EC00164 VJ=50.00
COMM MOVJ C00165 BC00165 VJ=50.00  +MOVJ EC00165 VJ=50.00
COMM MOVJ C00166 BC00166 VJ=50.00  +MOVJ EC00166 VJ=50.00
COMM MOVJ C00167 BC00167 VJ=50.00  +MOVJ EC00167 VJ=50.00
COMM MOVJ C00168 BC00168 VJ=50.00  +MOVJ EC00168 VJ=50.00
COMM SFTOF3D
COMM SMOVL C00169 BC00169 V=83.3  +MOVJ EC00169
COMM SREFP 3 C00170 BC00170  +REFP EC00170
COMM CALL JOB:SEARCH-R1-S13D
COMM SET P040 P006
COMM SFTON3D P040
COMM SMOVL C00171 BC00171 V=100.0  +MOVJ EC00171
COMM SMOVL C00172 BC00172 V=133.3  +MOVJ EC00172
COMM SMOVL C00173 BC00173 V=83.3 PL=0  +MOVJ EC00173
COMM SREFP 3 C00174 BC00174  +REFP EC00174
COMM CALL JOB:SEARCH-R1-S13D
COMM SET P040 P006
COMM SFTON3D P040
COMM SMOVL C00175 BC00175 V=100.0  +MOVJ EC00175
COMM SFTOF3D
COMM MACRO1 MJ#(0) ARGF9
COMM SFTON3D P040
COMM SMOVL C00176 BC00176 V=133.3  +MOVJ EC00176
COMM ARCON
COMM SMOVL C00177 BC00177 V=11.7  +MOVJ EC00177
COMM ARCOF
COMM MOVJ C00178 BC00178 VJ=20.00  +MOVJ EC00178 VJ=15.00
COMM MOVJ C00179 BC00179 VJ=30.00  +MOVJ EC00179 VJ=15.00
COMM 'SPAWDZIC CZY SPOINA TRAFIA
COMM SMOVL C00180 BC00180 V=166.7  +MOVJ EC00180
COMM ARCON
COMM SMOVL C00181 BC00181 V=12.5  +MOVJ EC00181
COMM ARCOF
COMM SMOVL C00182 BC00182 V=333.3  +MOVJ EC00182
COMM MOVJ C00183 BC00183 VJ=50.00  +MOVJ EC00183 VJ=50.00
COMM MOVJ C00184 BC00184 VJ=100.00  +MOVJ EC00184 VJ=50.00
COMM MOVJ C00185 BC00185 VJ=100.00  +MOVJ EC00185 VJ=50.00
COMM MOVJ C00186 BC00186 VJ=100.00  +MOVJ EC00186 VJ=50.00
COMM SFTON3D P040
COMM SMOVL C00187 BC00187 V=250.0  +MOVJ EC00187
COMM ARCON
COMM SMOVL C00188 BC00188 V=11.7  +MOVJ EC00188
COMM ARCOF
COMM SFTOF3D
COMM MOVJ C00189 BC00189 VJ=25.00  +MOVJ EC00189 VJ=50.00
COMM MOVJ C00190 BC00190 VJ=100.00  +MOVJ EC00190 VJ=50.00
COMM MOVJ C00191 BC00191 VJ=100.00  +MOVJ EC00191 VJ=50.00
COMM MOVJ C00192 BC00192 VJ=100.00  +MOVJ EC00192 VJ=50.00
COMM MOVJ C00193 BC00193 VJ=100.00  +MOVJ EC00193 VJ=50.00
COMM MOVJ C00194 BC00194 VJ=100.00  +MOVJ EC00194 VJ=50.00
COMM SFTOF3D
COMM MOVJ C00195 BC00195 VJ=100.00  +MOVJ EC00195 VJ=50.00
COMM SFTOF3D
COMM MOVJ C00196 BC00196 VJ=100.00  +MOVJ EC00196 VJ=50.00
COMM SFTON3D P041
COMM SMOVL C00197 BC00197 V=200.0  +MOVJ EC00197
COMM ARCON
COMM SMOVL C00198 BC00198 V=10.8  +MOVJ EC00198
COMM ARCOF
COMM SMOVL C00199 BC00199 V=83.3  +MOVJ EC00199
COMM ARCON
COMM SMOVL C00200 BC00200 V=10.0  +MOVJ EC00200
COMM ARCOF
COMM SMOVL C00201 BC00201 V=250.0  +MOVJ EC00201
COMM MOVJ C00202 BC00202 VJ=50.00  +MOVJ EC00202 VJ=50.00
COMM MOVJ C00203 BC00203 VJ=15.00  +MOVJ EC00203 VJ=50.00
COMM SMOVL C00204 BC00204 V=250.0  +MOVJ EC00204
COMM MACRO1 MJ#(0) ARGF9
COMM SMOVL C00205 BC00205 V=200.0  +MOVJ EC00205
COMM ARCON
COMM SMOVL C00206 BC00206 V=11.7  +MOVJ EC00206
COMM ARCOF
COMM SMOVL C00207 BC00207 V=333.3  +MOVJ EC00207
COMM SFTOF3D
COMM MOVJ C00208 BC00208 VJ=100.00  +MOVJ EC00208 VJ=50.00
COMM MOVJ C00209 BC00209 VJ=100.00  +MOVJ EC00209 VJ=50.00
COMM MOVJ C00210 BC00210 VJ=100.00  +MOVJ EC00210 VJ=50.00
COMM MOVJ C00211 BC00211 VJ=100.00  +MOVJ EC00211 VJ=50.00
COMM MOVJ C00212 BC00212 VJ=100.00  +MOVJ EC00212 VJ=50.00
COMM MOVJ C00213 BC00213 VJ=100.00  +MOVJ EC00213 VJ=50.00
COMM MOVJ C00214 BC00214 VJ=100.00  +MOVJ EC00214 VJ=50.00
COMM MOVJ C00215 BC00215 VJ=20.00  +MOVJ EC00215 VJ=50.00
COMM SFTON3D P040
COMM SMOVL C00216 BC00216 V=83.3  +MOVJ EC00216
COMM ARCON
COMM SMOVL C00217 BC00217 V=11.7  +MOVJ EC00217
COMM ARCOF
COMM SMOVL C00218 BC00218 V=133.3  +MOVJ EC00218
COMM SFTOF3D
COMM MOVJ C00219 BC00219 VJ=50.00  +MOVJ EC00219 VJ=50.00
COMM MOVJ C00220 BC00220 VJ=100.00  +MOVJ EC00220 VJ=50.00
COMM MOVJ C00221 BC00221 VJ=100.00  +MOVJ EC00221 VJ=50.00
COMM MOVJ C00222 BC00222 VJ=100.00  +MOVJ EC00222 VJ=50.00
COMM MOVJ C00223 BC00223 VJ=100.00  +MOVJ EC00223 VJ=50.00
COMM MOVJ C00224 BC00224 VJ=100.00  +MOVJ EC00224 VJ=50.00
COMM MOVJ C00225 BC00225 VJ=100.00  +MOVJ EC00225 VJ=50.00
COMM MOVJ C00226 BC00226 VJ=100.00  +MOVJ EC00226 VJ=50.00
COMM MOVJ C00227 BC00227 VJ=15.00  +MOVJ EC00227 VJ=50.00
COMM SFTON3D P041
COMM SMOVL C00228 BC00228 V=133.3  +MOVJ EC00228
COMM ARCON
COMM SMOVL C00229 BC00229 V=11.7  +MOVJ EC00229
COMM ARCOF
COMM SMOVL C00230 BC00230 V=133.3  +MOVJ EC00230
COMM SFTOF3D
COMM MOVJ C00231 BC00231 VJ=100.00  +MOVJ EC00231 VJ=50.00
COMM MOVJ C00232 BC00232 VJ=100.00  +MOVJ EC00232 VJ=50.00
COMM MOVJ C00233 BC00233 VJ=100.00  +MOVJ EC00233 VJ=50.00
COMM MOVJ C00234 BC00234 VJ=100.00  +MOVJ EC00234 VJ=50.00
COMM MOVJ C00235 BC00235 VJ=100.00  +MOVJ EC00235 VJ=50.00
COMM MOVJ C00236 BC00236 VJ=100.00  +MOVJ EC00236 VJ=50.00
COMM MOVJ C00237 BC00237 VJ=100.00  +MOVJ EC00237 VJ=50.00
COMM MOVJ C00238 BC00238 VJ=100.00  +MOVJ EC00238 VJ=50.00
COMM MOVJ C00239 BC00239 VJ=15.00  +MOVJ EC00239 VJ=50.00
COMM SFTON3D P040
COMM SMOVL C00240 BC00240 V=133.3  +MOVJ EC00240
COMM ARCON
COMM SMOVL C00241 BC00241 V=11.7  +MOVJ EC00241
COMM ARCOF
COMM SMOVL C00242 BC00242 V=133.3  +MOVJ EC00242
COMM MOVJ C00243 BC00243 VJ=100.00  +MOVJ EC00243 VJ=50.00
COMM MOVJ C00244 BC00244 VJ=100.00  +MOVJ EC00244 VJ=50.00
COMM MOVJ C00245 BC00245 VJ=100.00  +MOVJ EC00245 VJ=50.00
COMM MOVJ C00246 BC00246 VJ=15.00  +MOVJ EC00246 VJ=15.00
COMM SMOVL C00247 BC00247 V=133.3  +MOVJ EC00247
COMM ARCON
COMM SMOVL C00248 BC00248 V=11.7  +MOVJ EC00248
COMM ARCOF
COMM SMOVL C00249 BC00249 V=133.3  +MOVJ EC00249
COMM SMOVL C00250 BC00250 V=133.3  +MOVJ EC00250
COMM ARCON
COMM SMOVL C00251 BC00251 V=11.7  +MOVJ EC00251
COMM ARCOF
COMM SFTOF3D
COMM SMOVL C00252 BC00252 V=133.3  +MOVJ EC00252
COMM MOVJ C00253 BC00253 VJ=100.00  +MOVJ EC00253 VJ=50.00
COMM MOVJ C00254 BC00254 VJ=100.00  +MOVJ EC00254 VJ=50.00
COMM MOVJ C00255 BC00255 VJ=100.00  +MOVJ EC00255 VJ=50.00
COMM MOVJ C00256 BC00256 VJ=100.00  +MOVJ EC00256 VJ=50.00
COMM MOVJ C00257 BC00257 VJ=100.00  +MOVJ EC00257 VJ=50.00
COMM MOVJ C00258 BC00258 VJ=100.00  +MOVJ EC00258 VJ=50.00
COMM MOVJ C00259 BC00259 VJ=100.00  +MOVJ EC00259 VJ=50.00
COMM MOVJ C00260 BC00260 VJ=100.00  +MOVJ EC00260 VJ=50.00
COMM MOVJ C00261 BC00261 VJ=50.00  +MOVJ EC00261 VJ=50.00
COMM SFTON3D P041
COMM SMOVL C00262 BC00262 V=16.7  +MOVJ EC00262
COMM ARCON
COMM SMOVL C00263 BC00263 V=8.3  +MOVJ EC00263
COMM ARCOF
COMM SMOVL C00264 BC00264 V=250.0  +MOVJ EC00264
COMM MOVJ C00265 BC00265 VJ=100.00  +MOVJ EC00265 VJ=50.00
COMM MACRO1 MJ#(0) ARGF9
COMM SMOVL C00266 BC00266 V=250.0  +MOVJ EC00266
COMM ARCON
COMM SMOVL C00267 BC00267 V=11.7  +MOVJ EC00267
COMM SMOVL C00268 BC00268 V=11.7  +MOVJ EC00268
COMM ARCOF
COMM SMOVL C00269 BC00269 V=166.7  +MOVJ EC00269
COMM SMOVL C00270 BC00270 V=666.7  +MOVJ EC00270
COMM SMOVL C00271 BC00271 V=250.0  +MOVJ EC00271
COMM ARCON
COMM SMOVL C00272 BC00272 V=11.7  +MOVJ EC00272
COMM ARCOF
COMM SFTOF3D
COMM SMOVL C00273 BC00273 V=166.7  +MOVJ EC00273
COMM MOVJ C00274 BC00274 VJ=100.00  +MOVJ EC00274 VJ=50.00
COMM MOVJ C00275 BC00275 VJ=100.00  +MOVJ EC00275 VJ=50.00
COMM MOVJ C00276 BC00276 VJ=100.00  +MOVJ EC00276 VJ=50.00
COMM MOVJ C00277 BC00277 VJ=100.00  +MOVJ EC00277 VJ=50.00
COMM MOVJ C00278 BC00278 VJ=100.00  +MOVJ EC00278 VJ=50.00
COMM MOVJ C00279 BC00279 VJ=50.00  +MOVJ EC00279 VJ=50.00
COMM MOVJ C00280 BC00280 VJ=50.00  +MOVJ EC00280 VJ=50.00
COMM MOVJ C00281 BC00281 VJ=50.00  +MOVJ EC00281 VJ=50.00
COMM SFTON3D P040
COMM SMOVL C00282 BC00282 V=166.7  +MOVJ EC00282
COMM ARCON
COMM SMOVL C00283 BC00283 V=11.7  +MOVJ EC00283
COMM ARCOF
COMM SMOVL C00284 BC00284 V=333.3  +MOVJ EC00284
COMM SMOVL C00285 BC00285 V=666.7  +MOVJ EC00285
COMM SMOVL C00286 BC00286 V=166.7  +MOVJ EC00286
COMM ARCON
COMM SMOVL C00287 BC00287 V=11.7  +MOVJ EC00287
COMM ARCOF
COMM SMOVL C00288 BC00288 V=333.3  +MOVJ EC00288
COMM SFTOF3D
COMM MOVJ C00289 BC00289 VJ=50.00  +MOVJ EC00289 VJ=50.00
COMM MOVJ C00290 BC00290 VJ=50.00  +MOVJ EC00290 VJ=50.00
COMM MOVJ C00291 BC00291 VJ=50.00  +MOVJ EC00291 VJ=50.00
COMM MOVJ C00292 BC00292 VJ=50.00  +MOVJ EC00292 VJ=50.00
COMM MOVJ C00293 BC00293 VJ=50.00  +MOVJ EC00293 VJ=50.00
COMM MOVJ C00294 BC00294 VJ=100.00  +MOVJ EC00294 VJ=50.00
COMM MOVJ C00295 BC00295 VJ=100.00  +MOVJ EC00295 VJ=50.00
COMM MOVJ C00296 BC00296 VJ=50.00  +MOVJ EC00296 VJ=50.00
COMM SFTON3D P041
COMM SMOVL C00297 BC00297 V=250.0  +MOVJ EC00297
COMM ARCON
COMM SMOVL C00298 BC00298 V=11.7  +MOVJ EC00298
COMM ARCOF
COMM SMOVL C00299 BC00299 V=250.0  +MOVJ EC00299
COMM SMOVL C00300 BC00300 V=250.0  +MOVJ EC00300
COMM ARCON
COMM SMOVL C00301 BC00301 V=10.8  +MOVJ EC00301
COMM ARCOF
COMM SMOVL C00302 BC00302 V=250.0  +MOVJ EC00302
COMM SMOVL C00303 BC00303 V=666.7  +MOVJ EC00303
COMM MOVJ C00304 BC00304 VJ=100.00  +MOVJ EC00304 VJ=50.00
COMM SSFTOF
COMM MOVJ C00305 BC00305 VJ=100.00  +MOVJ EC00305 VJ=50.00
COMM CALL JOB:CLEAN-R1_KM2
COMM MOVJ C00306 BC00306 VJ=100.00  +MOVJ EC00306 VJ=50.00
COMM MOVJ C00307 BC00307 VJ=100.00  +MOVJ EC00307 VJ=15.00
COMM MOVJ C00308 BC00308 VJ=100.00  +MOVJ EC00308 VJ=50.00
COMM MOVJ C00309 BC00309 VJ=100.00  +MOVJ EC00309 VJ=50.00
COMM MOVJ C00310 BC00310 VJ=15.00  +MOVJ EC00310 VJ=15.00
COMM MOVJ C00311 BC00311 VJ=15.00  +MOVJ EC00311 VJ=50.00
COMM SMOVL C00312 BC00312 V=83.3  +MOVJ EC00312
COMM SREFP 3 C00313 BC00313  +REFP EC00313
COMM CALL JOB:SEARCH-R1-S13D
COMM SET P042 P006
COMM SFTON3D P042
COMM SMOVL C00314 BC00314 V=60.0  +MOVJ EC00314
COMM SMOVL C00315 BC00315 V=133.3  +MOVJ EC00315
COMM SMOVL C00316 BC00316 V=133.3  +MOVJ EC00316
COMM SREFP 3 C00317 BC00317  +REFP EC00317
COMM CALL JOB:SEARCH-R1-S13D
COMM SET P042 P006
COMM SFTON3D P042
COMM SMOVL C00318 BC00318 V=60.0  +MOVJ EC00318
COMM SFTOF3D
COMM MOVJ C00319 BC00319 VJ=15.00  +MOVJ EC00319 VJ=15.00
COMM MOVJ C00320 BC00320 VJ=15.00  +MOVJ EC00320 VJ=15.00
COMM MOVJ C00321 BC00321 VJ=15.00  +MOVJ EC00321 VJ=15.00
COMM MOVJ C00322 BC00322 VJ=15.00  +MOVJ EC00322 VJ=15.00
COMM SMOVL C00323 BC00323 V=83.3  +MOVJ EC00323
COMM SREFP 3 C00324 BC00324  +REFP EC00324
COMM CALL JOB:SEARCH-R1-S13D
COMM SET P043 P006
COMM SFTON3D P043
COMM SMOVL C00325 BC00325 V=60.0  +MOVJ EC00325
COMM SMOVL C00326 BC00326 V=133.3  +MOVJ EC00326
COMM SMOVL C00327 BC00327 V=133.3  +MOVJ EC00327
COMM SREFP 3 C00328 BC00328  +REFP EC00328
COMM CALL JOB:SEARCH-R1-S13D
COMM SET P043 P006
COMM SFTON3D P043
COMM SMOVL C00329 BC00329 V=60.0  +MOVJ EC00329
COMM MOVJ C00330 BC00330 VJ=30.00  +MOVJ EC00330 VJ=30.00
COMM SFTOF3D
COMM MOVJ C00331 BC00331 VJ=30.00  +MOVJ EC00331 VJ=30.00
COMM MOVJ C00332 BC00332 VJ=30.00  +MOVJ EC00332 VJ=30.00
COMM MOVJ C00333 BC00333 VJ=50.00  +MOVJ EC00333 VJ=50.00
COMM MOVJ C00334 BC00334 VJ=50.00  +MOVJ EC00334 VJ=50.00
COMM SFTOF3D
COMM MOVJ C00335 BC00335 VJ=30.00  +MOVJ EC00335 VJ=30.00
COMM SMOVL C00336 BC00336 V=83.3  +MOVJ EC00336
COMM SREFP 3 C00337 BC00337  +REFP EC00337
COMM CALL JOB:SEARCH-R1-S13D
COMM SET P044 P006
COMM SFTON3D P044
COMM SMOVL C00338 BC00338 V=100.0  +MOVJ EC00338
COMM SREFP 3 C00339 BC00339  +REFP EC00339
COMM CALL JOB:SEARCH-R1-S13D
COMM SET P044 P006
COMM SFTON3D P044
COMM SMOVL C00340 BC00340 V=133.3  +MOVJ EC00340
COMM SMOVL C00341 BC00341 V=250.0  +MOVJ EC00341
COMM SMOVL C00342 BC00342 V=133.3  +MOVJ EC00342
COMM SREFP 3 C00343 BC00343  +REFP EC00343
COMM CALL JOB:SEARCH-R1-S13D
COMM SET P044 P006
COMM SFTON3D P044
COMM SMOVL C00344 BC00344 V=133.3  +MOVJ EC00344
COMM SFTOF3D
COMM MOVJ C00345 BC00345 VJ=30.00  +MOVJ EC00345 VJ=15.00
COMM MOVJ C00346 BC00346 VJ=30.00  +MOVJ EC00346 VJ=15.00
COMM MOVJ C00347 BC00347 VJ=30.00  +MOVJ EC00347 VJ=15.00
COMM SMOVL C00348 BC00348 V=250.0  +MOVJ EC00348
COMM SREFP 3 C00349 BC00349  +REFP EC00349
COMM CALL JOB:SEARCH-R1-S13D
COMM SET P045 P006
COMM SFTON3D P045
COMM SMOVL C00350 BC00350 V=250.0  +MOVJ EC00350
COMM SREFP 3 C00351 BC00351  +REFP EC00351
COMM CALL JOB:SEARCH-R1-S13D
COMM SET P045 P006
COMM SFTON3D P045
COMM SMOVL C00352 BC00352 V=250.0  +MOVJ EC00352
COMM SMOVL C00353 BC00353 V=250.0  +MOVJ EC00353
COMM SMOVL C00354 BC00354 V=166.7  +MOVJ EC00354
COMM SREFP 3 C00355 BC00355  +REFP EC00355
COMM CALL JOB:SEARCH-R1-S13D
COMM SET P045 P006
COMM SFTON3D P045
COMM SMOVL C00356 BC00356 V=250.0  +MOVJ EC00356
COMM SFTOF3D
COMM MOVJ C00357 BC00357 VJ=30.00  +MOVJ EC00357 VJ=15.00
COMM MOVJ C00358 BC00358 VJ=30.00  +MOVJ EC00358 VJ=15.00
COMM SMOVL C00359 BC00359 V=250.0  +MOVJ EC00359
COMM SREFP 3 C00360 BC00360  +REFP EC00360
COMM CALL JOB:SEARCH-R1-S13D
COMM SET P046 P006
COMM SFTON3D P046
COMM SMOVL C00361 BC00361 V=250.0  +MOVJ EC00361
COMM SREFP 3 C00362 BC00362  +REFP EC00362
COMM CALL JOB:SEARCH-R1-S13D
COMM SET P046 P006
COMM SFTON3D P046
COMM SMOVL C00363 BC00363 V=250.0  +MOVJ EC00363
COMM SFTOF3D
COMM MOVJ C00364 BC00364 VJ=30.00  +MOVJ EC00364 VJ=15.00
COMM MOVJ C00365 BC00365 VJ=30.00  +MOVJ EC00365 VJ=15.00
COMM MOVJ C00366 BC00366 VJ=30.00  +MOVJ EC00366 VJ=15.00
COMM MOVJ C00367 BC00367 VJ=30.00  +MOVJ EC00367 VJ=15.00
COMM SMOVL C00368 BC00368 V=250.0  +MOVJ EC00368
COMM SREFP 3 C00369 BC00369  +REFP EC00369
COMM CALL JOB:SEARCH-R1-S13D
COMM SET P048 P006
COMM SFTON3D P048
COMM SMOVL C00370 BC00370 V=250.0  +MOVJ EC00370
COMM SREFP 3 C00371 BC00371  +REFP EC00371
COMM CALL JOB:SEARCH-R1-S13D
COMM SET P048 P006
COMM SFTON3D P048
COMM SMOVL C00372 BC00372 V=250.0  +MOVJ EC00372
COMM MOVJ C00373 BC00373 VJ=30.00  +MOVJ EC00373 VJ=15.00
COMM SFTOF3D
COMM MOVJ C00374 BC00374 VJ=30.00  +MOVJ EC00374 VJ=15.00
COMM MOVJ C00375 BC00375 VJ=30.00  +MOVJ EC00375 VJ=15.00
COMM SMOVL C00376 BC00376 V=166.7  +MOVJ EC00376
COMM SREFP 3 C00377 BC00377  +REFP EC00377
COMM CALL JOB:SEARCH-R1-S13D
COMM SET P049 P006
COMM SFTON3D P049
COMM SMOVL C00378 BC00378 V=166.7  +MOVJ EC00378
COMM SREFP 3 C00379 BC00379  +REFP EC00379
COMM CALL JOB:SEARCH-R1-S13D
COMM SET P049 P006
COMM SFTON3D P049
COMM SMOVL C00380 BC00380 V=166.7  +MOVJ EC00380
COMM SMOVL C00381 BC00381 V=166.7  +MOVJ EC00381
COMM SMOVL C00382 BC00382 V=166.7  +MOVJ EC00382
COMM SREFP 3 C00383 BC00383  +REFP EC00383
COMM CALL JOB:SEARCH-R1-S13D
COMM SET P049 P006
COMM SFTON3D P049
COMM SMOVL C00384 BC00384 V=166.7  +MOVJ EC00384
COMM SFTOF3D
COMM MOVJ C00385 BC00385 VJ=30.00  +MOVJ EC00385 VJ=30.00
COMM MOVJ C00386 BC00386 VJ=30.00  +MOVJ EC00386 VJ=30.00
COMM MOVJ C00387 BC00387 VJ=30.00  +MOVJ EC00387 VJ=15.00
COMM SMOVL C00388 BC00388 V=250.0  +MOVJ EC00388
COMM SREFP 3 C00389 BC00389  +REFP EC00389
COMM CALL JOB:SEARCH-R1-S13D
COMM SET P050 P006
COMM SFTON3D P050
COMM SMOVL C00390 BC00390 V=250.0  +MOVJ EC00390
COMM SREFP 3 C00391 BC00391  +REFP EC00391
COMM CALL JOB:SEARCH-R1-S13D
COMM SET P050 P006
COMM SFTON3D P050
COMM SMOVL C00392 BC00392 V=250.0  +MOVJ EC00392
COMM SMOVL C00393 BC00393 V=250.0  +MOVJ EC00393
COMM SMOVL C00394 BC00394 V=166.7  +MOVJ EC00394
COMM SREFP 3 C00395 BC00395  +REFP EC00395
COMM CALL JOB:SEARCH-R1-S13D
COMM SET P050 P006
COMM SFTON3D P050
COMM SMOVL C00396 BC00396 V=166.7  +MOVJ EC00396
COMM SFTOF3D
COMM MOVJ C00397 BC00397 VJ=30.00  +MOVJ EC00397 VJ=15.00
COMM MOVJ C00398 BC00398 VJ=30.00  +MOVJ EC00398 VJ=15.00
COMM MOVJ C00399 BC00399 VJ=30.00  +MOVJ EC00399 VJ=15.00
COMM MOVJ C00400 BC00400 VJ=30.00  +MOVJ EC00400 VJ=30.00
COMM MOVJ C00401 BC00401 VJ=30.00  +MOVJ EC00401 VJ=30.00
COMM MACRO1 MJ#(0) ARGF9
COMM SFTON3D P042
COMM SMOVL C00402 BC00402 V=166.7  +MOVJ EC00402
COMM ARCON
COMM SMOVC C00403 BC00403 V=8.3  +MOVJ EC00403
COMM SMOVC C00404 BC00404 V=8.3  +MOVJ EC00404
COMM SMOVC C00405 BC00405 V=8.3  +MOVJ EC00405
COMM SMOVL C00406 BC00406 V=8.3  +MOVJ EC00406
COMM ARCOF
COMM SFTOF3D
COMM SMOVL C00407 BC00407 V=250.0  +MOVJ EC00407
COMM SMOVL C00408 BC00408 V=250.0  +MOVJ EC00408
COMM SFTON3D P043
COMM SMOVL C00409 BC00409 V=166.7  +MOVJ EC00409
COMM ARCON
COMM SMOVC C00410 BC00410 V=8.3  +MOVJ EC00410
COMM SMOVC C00411 BC00411 V=8.3  +MOVJ EC00411
COMM SMOVC C00412 BC00412 V=8.3  +MOVJ EC00412
COMM SMOVL C00413 BC00413 V=8.3  +MOVJ EC00413
COMM ARCOF
COMM SFTOF3D
COMM SMOVL C00414 BC00414 V=166.7  +MOVJ EC00414
COMM SMOVL C00415 BC00415 V=250.0  +MOVJ EC00415
COMM MOVJ C00416 BC00416 VJ=30.00  +MOVJ EC00416 VJ=30.00
COMM MACRO1 MJ#(0) ARGF9
COMM MOVJ C00417 BC00417 VJ=15.00  +MOVJ EC00417 VJ=10.00
COMM SFTON3D P044
COMM SMOVL C00418 BC00418 V=166.7  +MOVJ EC00418
COMM ARCON
COMM SMOVL C00419 BC00419 V=9.2  +MOVJ EC00419
COMM SMOVL C00420 BC00420 V=9.2  +MOVJ EC00420
COMM ARCOF
COMM SFTOF3D
COMM SMOVL C00421 BC00421 V=250.0  +MOVJ EC00421
COMM SFTON3D P045
COMM SMOVL C00422 BC00422 V=166.7  +MOVJ EC00422
COMM ARCON
COMM SMOVL C00423 BC00423 V=9.2  +MOVJ EC00423
COMM SMOVL C00424 BC00424 V=9.2  +MOVJ EC00424
COMM ARCOF
COMM SMOVL C00425 BC00425 V=250.0  +MOVJ EC00425
COMM SFTON3D P046
COMM SMOVL C00426 BC00426 V=166.7  +MOVJ EC00426
COMM ARCON
COMM SMOVL C00427 BC00427 V=9.2  +MOVJ EC00427
COMM SMOVL C00428 BC00428 V=9.2  +MOVJ EC00428
COMM ARCOF
COMM SFTOF3D
COMM SMOVL C00429 BC00429 V=166.7  +MOVJ EC00429
COMM SMOVL C00430 BC00430 V=250.0  +MOVJ EC00430
COMM SMOVL C00431 BC00431 V=250.0  +MOVJ EC00431
COMM SMOVL C00432 BC00432 V=250.0  +MOVJ EC00432
COMM SFTON3D P045
COMM SMOVL C00433 BC00433 V=166.7  +MOVJ EC00433
COMM ARCON
COMM SMOVL C00434 BC00434 V=10.0  +MOVJ EC00434
COMM ARCOF
COMM SMOVL C00435 BC00435 V=250.0  +MOVJ EC00435
COMM SMOVL C00436 BC00436 V=333.3  +MOVJ EC00436
COMM SFTON3D P044
COMM SMOVL C00437 BC00437 V=166.7  +MOVJ EC00437
COMM ARCON
COMM SMOVL C00438 BC00438 V=10.0  +MOVJ EC00438
COMM ARCOF
COMM SMOVL C00439 BC00439 V=250.0  +MOVJ EC00439
COMM MOVJ C00440 BC00440 VJ=20.00  +MOVJ EC00440 VJ=10.00
COMM MOVJ C00441 BC00441 VJ=40.00  +MOVJ EC00441 VJ=10.00
COMM MOVJ C00442 BC00442 VJ=20.00  +MOVJ EC00442 VJ=10.00
COMM SFTON3D P050
COMM SMOVL C00443 BC00443 V=166.7  +MOVJ EC00443
COMM ARCON
COMM SMOVL C00444 BC00444 V=9.2  +MOVJ EC00444
COMM SMOVL C00445 BC00445 V=9.2  +MOVJ EC00445
COMM ARCOF
COMM SMOVL C00446 BC00446 V=166.7  +MOVJ EC00446
COMM SFTON3D P049
COMM SMOVL C00447 BC00447 V=166.7  +MOVJ EC00447
COMM ARCON
COMM SMOVL C00448 BC00448 V=9.2  +MOVJ EC00448
COMM SMOVL C00449 BC00449 V=9.2  +MOVJ EC00449
COMM SMOVL C00450 BC00450 V=9.2  +MOVJ EC00450
COMM ARCOF
COMM SMOVL C00451 BC00451 V=166.7  +MOVJ EC00451
COMM SFTON3D P048
COMM SMOVL C00452 BC00452 V=166.7  +MOVJ EC00452
COMM ARCON
COMM SMOVL C00453 BC00453 V=9.2  +MOVJ EC00453
COMM SMOVL C00454 BC00454 V=9.2  +MOVJ EC00454
COMM SMOVL C00455 BC00455 V=8.3  +MOVJ EC00455
COMM ARCOF
COMM SMOVL C00456 BC00456 V=166.7  +MOVJ EC00456
COMM SMOVL C00457 BC00457 V=166.7  +MOVJ EC00457
COMM SFTON3D P049
COMM SMOVL C00458 BC00458 V=166.7  +MOVJ EC00458
COMM ARCON
COMM SMOVL C00459 BC00459 V=10.0  +MOVJ EC00459
COMM ARCOF
COMM SMOVL C00460 BC00460 V=250.0  +MOVJ EC00460
COMM SFTON3D P050
COMM SMOVL C00461 BC00461 V=200.0  +MOVJ EC00461
COMM ARCON
COMM SMOVL C00462 BC00462 V=10.0  +MOVJ EC00462
COMM ARCOF
COMM SFTOF3D
COMM SMOVL C00463 BC00463 V=250.0  +MOVJ EC00463
COMM MOVJ C00464 BC00464 VJ=60.00  +MOVJ EC00464 VJ=60.00
COMM MOVJ C00465 BC00465 VJ=60.00  +MOVJ EC00465 VJ=60.00
COMM MOVJ C00466 BC00466 VJ=60.00  +MOVJ EC00466 VJ=60.00
COMM MOVJ C00467 BC00467 VJ=100.00  +MOVJ EC00467 VJ=100.00
END
